LIN {X 0,Y 169.954,Z 453.379,A -85,B 0,C 180,E1 -25767.886,E2 -25767.886} C_VEL
LIN {X 0,Y 165.265,Z 466.004,A -85,B 0,C 180,E1 -25769.338,E2 -25769.338} C_VEL
LIN {X 0,Y 160.143,Z 477.221,A -85,B 0,C 180,E1 -25771.158,E2 -25771.158} C_VEL
LIN {X 0,Y 154.638,Z 487.355,A -85,B 0,C 180,E1 -25773.432,E2 -25773.432} C_VEL
LIN {X 0,Y 148.228,Z 497.15,A -85,B 0,C 180,E1 -25776.293,E2 -25776.293} C_VEL
LIN {X 0,Y 142.57,Z 504.593,A -85,B 0,C 180,E1 -25779.183,E2 -25779.183} C_VEL
LIN {X 0,Y 136.506,Z 511.591,A -85,B 0,C 180,E1 -25782.809,E2 -25782.809} C_VEL
LIN {X 0,Y 129.978,Z 518.044,A -85,B 0,C 180,E1 -25787.48,E2 -25787.48} C_VEL
LIN {X 0,Y 125.036,Z 522.318,A -85,B 0,C 180,E1 -25791.9,E2 -25791.9} C_VEL
LIN {X 0,Y 122.256,Z 524.487,A -85,B 0,C 180,E1 -25794.913,E2 -25794.913} C_VEL
LIN {X 0,Y 119.731,Z 526.212,A -85,B 0,C 180,E1 -25798.113,E2 -25798.113} C_VEL
LIN {X 0,Y 115.834,Z 528.4,A -85,B 0,C 180,E1 -25804.87,E2 -25804.87} C_VEL
LIN {X 0,Y 114.432,Z 528.886,A -85,B 0,C 180,E1 -25808.379,E2 -25808.379} C_VEL
LIN {X 0,Y 113.36,Z 528.935,A -85,B 0,C 180,E1 -25811.944,E2 -25811.944} C_VEL
LIN {X 0,Y 112.313,Z 527.87,A -85,B 0,C 180,E1 -25819.182,E2 -25819.182} C_VEL
LIN {X 0,Y 112.317,Z 526.734,A -85,B 0,C 180,E1 -25822.813,E2 -25822.813} C_VEL
LIN {X 0,Y 112.709,Z 525.151,A -85,B 0,C 180,E1 -25826.427,E2 -25826.427} C_VEL
LIN {X 0,Y 113.499,Z 522.024,A -85,B 0,C 180,E1 -25831.776,E2 -25831.776} C_VEL
LIN {X 0,Y 115.038,Z 517.849,A -85,B 0,C 180,E1 -25837.021,E2 -25837.021} C_VEL
LIN {X 0,Y 117.816,Z 511.498,A -85,B 0,C 180,E1 -25842.928,E2 -25842.928} C_VEL
LIN {X 0,Y 120.909,Z 504.594,A -85,B 0,C 180,E1 -25847.77,E2 -25847.77} C_VEL
LIN {X 0,Y 124.835,Z 495.925,A -85,B 0,C 180,E1 -25852.337,E2 -25852.337} C_VEL
LIN {X 0,Y 128.597,Z 487.054,A -85,B 0,C 180,E1 -25855.928,E2 -25855.928} C_VEL
LIN {X 0,Y 132.376,Z 477.3,A -85,B 0,C 180,E1 -25858.979,E2 -25858.979} C_VEL
LIN {X 0,Y 136.006,Z 466.57,A -85,B 0,C 180,E1 -25861.55,E2 -25861.55} C_VEL
LIN {X 0,Y 139.168,Z 454.593,A -85,B 0,C 180,E1 -25863.747,E2 -25863.747} C_VEL
LIN {X 0,Y 141.844,Z 442.071,A -85,B 0,C 180,E1 -25865.388,E2 -25865.388} C_VEL
LIN {X 0,Y 143.68,Z 429.753,A -85,B 0,C 180,E1 -25866.505,E2 -25866.505} C_VEL
LIN {X 0,Y 144.953,Z 414.737,A -85,B 0,C 180,E1 -25867.3,E2 -25867.3} C_VEL
LIN {X 0,Y 147.183,Z 381.844,A -85,B 0,C 180,E1 -25868.662,E2 -25868.662} C_VEL
LIN {X 0,Y 143.364,Z 373.581,A -85,B 0,C 180,E1 -25870.727,E2 -25870.727} C_VEL
LIN {X 0,Y 138.443,Z 364.416,A -85,B 0,C 180,E1 -25873.568,E2 -25873.568} C_VEL
LIN {X 0,Y 132.527,Z 354.94,A -85,B 0,C 180,E1 -25877.383,E2 -25877.383} C_VEL
LIN {X 0,Y 129.11,Z 350.145,A -85,B 0,C 180,E1 -25879.855,E2 -25879.855} C_VEL
LIN {X 0,Y 126.584,Z 346.535,A -85,B 0,C 180,E1 -25881.884,E2 -25881.884} C_VEL
LIN {X 0,Y 124.126,Z 343.341,A -85,B 0,C 180,E1 -25884.023,E2 -25884.023} C_VEL
LIN {X 0,Y 123.216,Z 342.017,A -85,B 0,C 180,E1 -25884.889,E2 -25884.889} C_VEL
LIN {X 0,Y 120.836,Z 339.591,A -85,B 0,C 180,E1 -25887.204,E2 -25887.204} C_VEL
LIN {X 0,Y 119.433,Z 336.949,A -85,B 0,C 180,E1 -25888.862,E2 -25888.862} C_VEL
LIN {X 0,Y 116.762,Z 335.135,A -85,B 0,C 180,E1 -25891.949,E2 -25891.949} C_VEL
LIN {X 0,Y 115.281,Z 332.838,A -85,B 0,C 180,E1 -25894.132,E2 -25894.132} C_VEL
LIN {X 0,Y 114.896,Z 331.137,A -85,B 0,C 180,E1 -25895.066,E2 -25895.066} C_VEL
LIN {X 0,Y 114.985,Z 331.156,A -85,B 0,C 180,E1 -25898.485,E2 -25898.485} C_VEL
LIN {X 0,Y 115.113,Z 331.108,A -85,B 0,C 180,E1 -25905.864,E2 -25905.864} C_VEL
LIN {X 0,Y 115.315,Z 331.119,A -85,B 0,C 180,E1 -25909.464,E2 -25909.464} C_VEL
LIN {X 0,Y 115.489,Z 331.058,A -85,B 0,C 180,E1 -25916.51,E2 -25916.51} C_VEL
LIN {X 0,Y 115.977,Z 331.035,A -85,B 0,C 180,E1 -25919.999,E2 -25919.999} C_VEL
LIN {X 0,Y 115.35,Z 331.075,A -85,B 0,C 180,E1 -25926.998,E2 -25926.998} C_VEL
LIN {X 0,Y 115.209,Z 331.131,A -85,B 0,C 180,E1 -25932.558,E2 -25932.558} C_VEL
LIN {X 0,Y 115.029,Z 331.167,A -85,B 0,C 180,E1 -25935.617,E2 -25935.617} C_VEL
LIN {X 0,Y 115.766,Z 333.599,A -85,B 0,C 180,E1 -25936.987,E2 -25936.987} C_VEL
LIN {X 0,Y 117.399,Z 335.687,A -85,B 0,C 180,E1 -25939.223,E2 -25939.223} C_VEL
LIN {X 0,Y 119.578,Z 337.12,A -85,B 0,C 180,E1 -25941.67,E2 -25941.67} C_VEL
LIN {X 0,Y 121.212,Z 340.163,A -85,B 0,C 180,E1 -25943.566,E2 -25943.566} C_VEL
LIN {X 0,Y 123.785,Z 342.605,A -85,B 0,C 180,E1 -25945.991,E2 -25945.991} C_VEL
LIN {X 0,Y 126.065,Z 346.012,A -85,B 0,C 180,E1 -25948.058,E2 -25948.058} C_VEL
LIN {X 0,Y 127.461,Z 347.601,A -85,B 0,C 180,E1 -25949.184,E2 -25949.184} C_VEL
LIN {X 0,Y 132.939,Z 355.533,A -85,B 0,C 180,E1 -25953.263,E2 -25953.263} C_VEL
LIN {X 0,Y 135.888,Z 360.462,A -85,B 0,C 180,E1 -25955.238,E2 -25955.238} C_VEL
LIN {X 0,Y 140.904,Z 371.644,A -85,B 0,C 180,E1 -25958.455,E2 -25958.455} C_VEL
LIN {X 0,Y 144.8,Z 382.281,A -85,B 0,C 180,E1 -25960.822,E2 -25960.822} C_VEL
LIN {X 0,Y 145.866,Z 386.133,A -85,B 0,C 180,E1 -25961.495,E2 -25961.495} C_VEL
LIN {X 0,Y 146.293,Z 398.588,A -85,B 0,C 180,E1 -25962.485,E2 -25962.485} C_VEL
LIN {X 0,Y 143.56,Z 436.22,A -85,B 0,C 180,E1 -25964.112,E2 -25964.112} C_VEL
LIN {X 0,Y 141.608,Z 449.705,A -85,B 0,C 180,E1 -25965.163,E2 -25965.163} C_VEL
LIN {X 0,Y 138.867,Z 462.391,A -85,B 0,C 180,E1 -25966.652,E2 -25966.652} C_VEL
LIN {X 0,Y 135.486,Z 474.2,A -85,B 0,C 180,E1 -25968.593,E2 -25968.593} C_VEL
LIN {X 0,Y 131.576,Z 485.585,A -85,B 0,C 180,E1 -25971.123,E2 -25971.123} C_VEL
LIN {X 0,Y 127.594,Z 495.844,A -85,B 0,C 180,E1 -25974.178,E2 -25974.178} C_VEL
LIN {X 0,Y 123.397,Z 505.909,A -85,B 0,C 180,E1 -25978.206,E2 -25978.206} C_VEL
LIN {X 0,Y 120.567,Z 511.911,A -85,B 0,C 180,E1 -25981.194,E2 -25981.194} C_VEL
LIN {X 0,Y 118.406,Z 517.269,A -85,B 0,C 180,E1 -25984.51,E2 -25984.51} C_VEL
LIN {X 0,Y 116.081,Z 522.835,A -85,B 0,C 180,E1 -25988.697,E2 -25988.697} C_VEL
LIN {X 0,Y 113.916,Z 528.259,A -85,B 0,C 180,E1 -25993.879,E2 -25993.879} C_VEL
LIN {X 0,Y 112.782,Z 532.492,A -85,B 0,C 180,E1 -25999.223,E2 -25999.223} C_VEL
LIN {X 0,Y 112.433,Z 534.724,A -85,B 0,C 180,E1 -26002.816,E2 -26002.816} C_VEL
LIN {X 0,Y 112.492,Z 537.26,A -85,B 0,C 180,E1 -26008.387,E2 -26008.387} C_VEL
LIN {X 0,Y 112.47,Z 538.122,A -85,B 0,C 180,E1 -26011.162,E2 -26011.162} C_VEL
LIN {X 0,Y 112.405,Z 539.12,A -85,B 0,C 180,E1 -26017.181,E2 -26017.181} C_VEL
LIN {X 0,Y 113.531,Z 538.827,A -85,B 0,C 180,E1 -26024.334,E2 -26024.334} C_VEL
LIN {X 0,Y 116.284,Z 537.016,A -85,B 0,C 180,E1 -26031.259,E2 -26031.259} C_VEL
LIN {X 0,Y 118.375,Z 535.488,A -85,B 0,C 180,E1 -26034.554,E2 -26034.554} C_VEL
LIN {X 0,Y 122.165,Z 532.423,A -85,B 0,C 180,E1 -26039.272,E2 -26039.272} C_VEL
LIN {X 0,Y 126.661,Z 528.327,A -85,B 0,C 180,E1 -26043.699,E2 -26043.699} C_VEL
LIN {X 0,Y 132.806,Z 522.078,A -85,B 0,C 180,E1 -26048.445,E2 -26048.445} C_VEL
LIN {X 0,Y 138.861,Z 515.309,A -85,B 0,C 180,E1 -26052.111,E2 -26052.111} C_VEL
LIN {X 0,Y 145.542,Z 506.936,A -85,B 0,C 180,E1 -26055.416,E2 -26055.416} C_VEL
LIN {X 0,Y 151.382,Z 498.339,A -85,B 0,C 180,E1 -26057.969,E2 -26057.969} C_VEL
LIN {X 0,Y 153.654,Z 494.853,A -85,B 0,C 180,E1 -26058.768,E2 -26058.768} C_VEL
LIN {X 0,Y 155.897,Z 490.401,A -85,B 0,C 180,E1 -26059.955,E2 -26059.955} C_VEL
LIN {X 0,Y 158.231,Z 482.914,A -85,B 0,C 180,E1 -26062.187,E2 -26062.187} C_VEL
LIN {X 0,Y 160.346,Z 474.972,A -85,B 0,C 180,E1 -26064.172,E2 -26064.172} C_VEL
LIN {X 0,Y 162.147,Z 469.815,A -85,B 0,C 180,E1 -26064.959,E2 -26064.959} C_VEL
LIN {X 0,Y 166.612,Z 457.272,A -85,B 0,C 180,E1 -26066.142,E2 -26066.142} C_VEL
LIN {X 0,Y 169.968,Z 444.445,A -85,B 0,C 180,E1 -26066.992,E2 -26066.992} C_VEL
LIN {X 0,Y 172.089,Z 431.144,A -85,B 0,C 180,E1 -26067.598,E2 -26067.598} C_VEL
LIN {X 0,Y 173.3,Z 418.29,A -85,B 0,C 180,E1 -26068.013,E2 -26068.013} C_VEL
LIN {X 0,Y 170.042,Z 408.838,A -85,B 0,C 180,E1 -26071.06,E2 -26071.06} C_VEL
LIN {X 0,Y 166.847,Z 400.851,A -85,B 0,C 180,E1 -26074.424,E2 -26074.424} C_VEL
LIN {X 0,Y 164.442,Z 395.255,A -85,B 0,C 180,E1 -26077.379,E2 -26077.379} C_VEL
LIN {X 0,Y 161.996,Z 390.005,A -85,B 0,C 180,E1 -26081.012,E2 -26081.012} C_VEL
LIN {X 0,Y 159.926,Z 386.674,A -85,B 0,C 180,E1 -26084.859,E2 -26084.859} C_VEL
LIN {X 0,Y 159.509,Z 385.905,A -85,B 0,C 180,E1 -26085.846,E2 -26085.846} C_VEL
LIN {X 0,Y 157.79,Z 383.124,A -85,B 0,C 180,E1 -26091.856,E2 -26091.856} C_VEL
LIN {X 0,Y 157.642,Z 381.317,A -85,B 0,C 180,E1 -26094.885,E2 -26094.885} C_VEL
LIN {X 0,Y 157.697,Z 381.298,A -85,B 0,C 180,E1 -26097.59,E2 -26097.59} C_VEL
LIN {X 0,Y 158.291,Z 384.205,A -85,B 0,C 180,E1 -26102.307,E2 -26102.307} C_VEL
LIN {X 0,Y 159.882,Z 386.192,A -85,B 0,C 180,E1 -26106.627,E2 -26106.627} C_VEL
LIN {X 0,Y 161.996,Z 389.909,A -85,B 0,C 180,E1 -26110.649,E2 -26110.649} C_VEL
LIN {X 0,Y 165.028,Z 395.159,A -85,B 0,C 180,E1 -26114.884,E2 -26114.884} C_VEL
LIN {X 0,Y 168.167,Z 400.686,A -85,B 0,C 180,E1 -26118.346,E2 -26118.346} C_VEL
LIN {X 0,Y 172.368,Z 408.93,A -85,B 0,C 180,E1 -26122.237,E2 -26122.237} C_VEL
LIN {X 0,Y 173.842,Z 412.055,A -85,B 0,C 180,E1 -26123.463,E2 -26123.463} C_VEL
LIN {X 0,Y 171.856,Z 429.918,A -85,B 0,C 180,E1 -26124.078,E2 -26124.078} C_VEL
LIN {X 0,Y 169.4,Z 442.515,A -85,B 0,C 180,E1 -26124.856,E2 -26124.856} C_VEL
LIN {X 0,Y 165.916,Z 454.623,A -85,B 0,C 180,E1 -26125.912,E2 -26125.912} C_VEL
LIN {X 0,Y 161.171,Z 466.872,A -85,B 0,C 180,E1 -26127.322,E2 -26127.322} C_VEL
LIN {X 0,Y 155.877,Z 477.959,A -85,B 0,C 180,E1 -26129.129,E2 -26129.129} C_VEL
LIN {X 0,Y 150.482,Z 487.489,A -85,B 0,C 180,E1 -26131.254,E2 -26131.254} C_VEL
LIN {X 0,Y 144.072,Z 496.935,A -85,B 0,C 180,E1 -26133.979,E2 -26133.979} C_VEL
LIN {X 0,Y 138.219,Z 504.334,A -85,B 0,C 180,E1 -26136.793,E2 -26136.793} C_VEL
LIN {X 0,Y 132.466,Z 510.715,A -85,B 0,C 180,E1 -26139.988,E2 -26139.988} C_VEL
LIN {X 0,Y 126.633,Z 516.425,A -85,B 0,C 180,E1 -26143.826,E2 -26143.826} C_VEL
LIN {X 0,Y 121.169,Z 521.105,A -85,B 0,C 180,E1 -26148.165,E2 -26148.165} C_VEL
LIN {X 0,Y 116.381,Z 524.643,A -85,B 0,C 180,E1 -26152.855,E2 -26152.855} C_VEL
LIN {X 0,Y 113.63,Z 526.425,A -85,B 0,C 180,E1 -26156.178,E2 -26156.178} C_VEL
LIN {X 0,Y 109.315,Z 528.668,A -85,B 0,C 180,E1 -26163.256,E2 -26163.256} C_VEL
LIN {X 0,Y 107.754,Z 529.194,A -85,B 0,C 180,E1 -26166.965,E2 -26166.965} C_VEL
LIN {X 0,Y 106.525,Z 529.284,A -85,B 0,C 180,E1 -26170.741,E2 -26170.741} C_VEL
LIN {X 0,Y 105.254,Z 528.274,A -85,B 0,C 180,E1 -26178.447,E2 -26178.447} C_VEL
LIN {X 0,Y 105.214,Z 527.182,A -85,B 0,C 180,E1 -26182.325,E2 -26182.325} C_VEL
LIN {X 0,Y 105.622,Z 525.499,A -85,B 0,C 180,E1 -26186.473,E2 -26186.473} C_VEL
LIN {X 0,Y 106.413,Z 522.565,A -85,B 0,C 180,E1 -26191.895,E2 -26191.895} C_VEL
LIN {X 0,Y 107.983,Z 518.455,A -85,B 0,C 180,E1 -26197.482,E2 -26197.482} C_VEL
LIN {X 0,Y 110.91,Z 512.171,A -85,B 0,C 180,E1 -26203.749,E2 -26203.749} C_VEL
LIN {X 0,Y 114.193,Z 505.347,A -85,B 0,C 180,E1 -26208.853,E2 -26208.853} C_VEL
LIN {X 0,Y 118.337,Z 496.805,A -85,B 0,C 180,E1 -26213.636,E2 -26213.636} C_VEL
LIN {X 0,Y 122.271,Z 488.046,A -85,B 0,C 180,E1 -26217.379,E2 -26217.379} C_VEL
LIN {X 0,Y 126.71,Z 477.255,A -85,B 0,C 180,E1 -26220.87,E2 -26220.87} C_VEL
LIN {X 0,Y 130.528,Z 466.399,A -85,B 0,C 180,E1 -26223.499,E2 -26223.499} C_VEL
LIN {X 0,Y 133.872,Z 454.288,A -85,B 0,C 180,E1 -26225.737,E2 -26225.737} C_VEL
LIN {X 0,Y 136.679,Z 441.562,A -85,B 0,C 180,E1 -26227.404,E2 -26227.404} C_VEL
LIN {X 0,Y 138.605,Z 428.722,A -85,B 0,C 180,E1 -26228.527,E2 -26228.527} C_VEL
LIN {X 0,Y 140.024,Z 411.792,A -85,B 0,C 180,E1 -26229.383,E2 -26229.383} C_VEL
LIN {X 0,Y 141.986,Z 384.117,A -85,B 0,C 180,E1 -26230.548,E2 -26230.548} C_VEL
LIN {X 0,Y 136.478,Z 372.568,A -85,B 0,C 180,E1 -26233.867,E2 -26233.867} C_VEL
LIN {X 0,Y 131.079,Z 363.313,A -85,B 0,C 180,E1 -26237.464,E2 -26237.464} C_VEL
LIN {X 0,Y 126.527,Z 356.335,A -85,B 0,C 180,E1 -26240.933,E2 -26240.933} C_VEL
LIN {X 0,Y 123.686,Z 352.328,A -85,B 0,C 180,E1 -26243.37,E2 -26243.37} C_VEL
LIN {X 0,Y 120.776,Z 348.238,A -85,B 0,C 180,E1 -26246.188,E2 -26246.188} C_VEL
LIN {X 0,Y 118.216,Z 345.2,A -85,B 0,C 180,E1 -26248.944,E2 -26248.944} C_VEL
LIN {X 0,Y 117.162,Z 343.409,A -85,B 0,C 180,E1 -26250.275,E2 -26250.275} C_VEL
LIN {X 0,Y 114.737,Z 341.346,A -85,B 0,C 180,E1 -26253.389,E2 -26253.389} C_VEL
LIN {X 0,Y 113.179,Z 338.5,A -85,B 0,C 180,E1 -26256.004,E2 -26256.004} C_VEL
LIN {X 0,Y 112.812,Z 337.909,A -85,B 0,C 180,E1 -26256.666,E2 -26256.666} C_VEL
LIN {X 0,Y 109.796,Z 335.963,A -85,B 0,C 180,E1 -26262.779,E2 -26262.779} C_VEL
LIN {X 0,Y 108.452,Z 333.244,A -85,B 0,C 180,E1 -26267.91,E2 -26267.91} C_VEL
LIN {X 0,Y 108.274,Z 331.996,A -85,B 0,C 180,E1 -26269.716,E2 -26269.716} C_VEL
LIN {X 0,Y 108.902,Z 331.915,A -85,B 0,C 180,E1 -26279.999,E2 -26279.999} C_VEL
LIN {X 0,Y 108.583,Z 332.143,A -85,B 0,C 180,E1 -26282.433,E2 -26282.433} C_VEL
LIN {X 0,Y 108.955,Z 334.021,A -85,B 0,C 180,E1 -26284.624,E2 -26284.624} C_VEL
LIN {X 0,Y 111.057,Z 336.803,A -85,B 0,C 180,E1 -26290.482,E2 -26290.482} C_VEL
LIN {X 0,Y 113.226,Z 338.186,A -85,B 0,C 180,E1 -26294.375,E2 -26294.375} C_VEL
LIN {X 0,Y 114.698,Z 341.256,A -85,B 0,C 180,E1 -26296.92,E2 -26296.92} C_VEL
LIN {X 0,Y 117.543,Z 343.903,A -85,B 0,C 180,E1 -26300.564,E2 -26300.564} C_VEL
LIN {X 0,Y 119.702,Z 347.229,A -85,B 0,C 180,E1 -26303.098,E2 -26303.098} C_VEL
LIN {X 0,Y 121.442,Z 349.031,A -85,B 0,C 180,E1 -26304.835,E2 -26304.835} C_VEL
LIN {X 0,Y 124.045,Z 352.644,A -85,B 0,C 180,E1 -26307.294,E2 -26307.294} C_VEL
LIN {X 0,Y 128.199,Z 358.783,A -85,B 0,C 180,E1 -26310.755,E2 -26310.755} C_VEL
LIN {X 0,Y 131.886,Z 364.746,A -85,B 0,C 180,E1 -26313.477,E2 -26313.477} C_VEL
LIN {X 0,Y 136.397,Z 375.036,A -85,B 0,C 180,E1 -26316.653,E2 -26316.653} C_VEL
LIN {X 0,Y 140.213,Z 385.883,A -85,B 0,C 180,E1 -26319.199,E2 -26319.199} C_VEL
LIN {X 0,Y 140.883,Z 388.479,A -85,B 0,C 180,E1 -26319.67,E2 -26319.67} C_VEL
LIN {X 0,Y 141.103,Z 399.609,A -85,B 0,C 180,E1 -26320.555,E2 -26320.555} C_VEL
LIN {X 0,Y 138.379,Z 435.693,A -85,B 0,C 180,E1 -26322.145,E2 -26322.145} C_VEL
LIN {X 0,Y 136.308,Z 449.382,A -85,B 0,C 180,E1 -26323.218,E2 -26323.218} C_VEL
LIN {X 0,Y 133.493,Z 461.901,A -85,B 0,C 180,E1 -26324.703,E2 -26324.703} C_VEL
LIN {X 0,Y 130.223,Z 472.946,A -85,B 0,C 180,E1 -26326.517,E2 -26326.517} C_VEL
LIN {X 0,Y 126.133,Z 484.507,A -85,B 0,C 180,E1 -26329.101,E2 -26329.101} C_VEL
LIN {X 0,Y 121.913,Z 494.927,A -85,B 0,C 180,E1 -26332.227,E2 -26332.227} C_VEL
LIN {X 0,Y 118.145,Z 503.441,A -85,B 0,C 180,E1 -26335.587,E2 -26335.587} C_VEL
LIN {X 0,Y 113.695,Z 512.647,A -85,B 0,C 180,E1 -26340.36,E2 -26340.36} C_VEL
LIN {X 0,Y 111.401,Z 517.812,A -85,B 0,C 180,E1 -26343.791,E2 -26343.791} C_VEL
LIN {X 0,Y 108.521,Z 524.19,A -85,B 0,C 180,E1 -26349.131,E2 -26349.131} C_VEL
LIN {X 0,Y 106.527,Z 529.254,A -85,B 0,C 180,E1 -26354.696,E2 -26354.696} C_VEL
LIN {X 0,Y 105.532,Z 533.167,A -85,B 0,C 180,E1 -26360.414,E2 -26360.414} C_VEL
LIN {X 0,Y 105.32,Z 536.026,A -85,B 0,C 180,E1 -26366.171,E2 -26366.171} C_VEL
LIN {X 0,Y 105.431,Z 537.605,A -85,B 0,C 180,E1 -26370.856,E2 -26370.856} C_VEL
LIN {X 0,Y 105.334,Z 538.761,A -85,B 0,C 180,E1 -26377.666,E2 -26377.666} C_VEL
LIN {X 0,Y 105.769,Z 538.844,A -85,B 0,C 180,E1 -26381.496,E2 -26381.496} C_VEL
LIN {X 0,Y 107.904,Z 537.837,A -85,B 0,C 180,E1 -26389.003,E2 -26389.003} C_VEL
LIN {X 0,Y 109.684,Z 536.767,A -85,B 0,C 180,E1 -26392.607,E2 -26392.607} C_VEL
LIN {X 0,Y 111.941,Z 535.286,A -85,B 0,C 180,E1 -26396.068,E2 -26396.068} C_VEL
LIN {X 0,Y 116.011,Z 532.268,A -85,B 0,C 180,E1 -26400.99,E2 -26400.99} C_VEL
LIN {X 0,Y 120.794,Z 528.222,A -85,B 0,C 180,E1 -26405.576,E2 -26405.576} C_VEL
LIN {X 0,Y 127.306,Z 522.046,A -85,B 0,C 180,E1 -26410.439,E2 -26410.439} C_VEL
LIN {X 0,Y 133.678,Z 515.346,A -85,B 0,C 180,E1 -26414.153,E2 -26414.153} C_VEL
LIN {X 0,Y 140.657,Z 507.06,A -85,B 0,C 180,E1 -26417.473,E2 -26417.473} C_VEL
LIN {X 0,Y 146.735,Z 498.585,A -85,B 0,C 180,E1 -26420.023,E2 -26420.023} C_VEL
LIN {X 0,Y 153.27,Z 488.129,A -85,B 0,C 180,E1 -26422.274,E2 -26422.274} C_VEL
LIN {X 0,Y 159.292,Z 476.387,A -85,B 0,C 180,E1 -26424.162,E2 -26424.162} C_VEL
LIN {X 0,Y 162.147,Z 469.815,A -85,B 0,C 180,E1 -26424.959,E2 -26424.959} C_VEL
LIN {X 0,Y 163.869,Z 464.575,A -85,B 0,C 180,E1 -26425.674,E2 -26425.674} C_VEL
LIN {X 0,Y 165.34,Z 455.878,A -85,B 0,C 180,E1 -26427.273,E2 -26427.273} C_VEL
LIN {X 0,Y 166.335,Z 446.985,A -85,B 0,C 180,E1 -26428.752,E2 -26428.752} C_VEL
LIN {X 0,Y 167.207,Z 441.344,A -85,B 0,C 180,E1 -26429.277,E2 -26429.277} C_VEL
LIN {X 0,Y 169.186,Z 428.054,A -85,B 0,C 180,E1 -26429.805,E2 -26429.805} C_VEL
LIN {X 0,Y 169.798,Z 421.095,A -85,B 0,C 180,E1 -26430.049,E2 -26430.049} C_VEL
LIN {X 0,Y 167.122,Z 413.122,A -85,B 0,C 180,E1 -26432.835,E2 -26432.835} C_VEL
LIN {X 0,Y 164.516,Z 406.154,A -85,B 0,C 180,E1 -26435.899,E2 -26435.899} C_VEL
LIN {X 0,Y 162.539,Z 401.124,A -85,B 0,C 180,E1 -26438.604,E2 -26438.604} C_VEL
LIN {X 0,Y 160.748,Z 396.858,A -85,B 0,C 180,E1 -26441.521,E2 -26441.521} C_VEL
LIN {X 0,Y 158.687,Z 393.329,A -85,B 0,C 180,E1 -26445.628,E2 -26445.628} C_VEL
LIN {X 0,Y 156.786,Z 389.519,A -85,B 0,C 180,E1 -26453.162,E2 -26453.162} C_VEL
LIN {X 0,Y 156.768,Z 388.418,A -85,B 0,C 180,E1 -26454.857,E2 -26454.857} C_VEL
LIN {X 0,Y 156.798,Z 388.676,A -85,B 0,C 180,E1 -26457.721,E2 -26457.721} C_VEL
LIN {X 0,Y 157.349,Z 391.227,A -85,B 0,C 180,E1 -26462.08,E2 -26462.08} C_VEL
LIN {X 0,Y 158.686,Z 392.968,A -85,B 0,C 180,E1 -26465.959,E2 -26465.959} C_VEL
LIN {X 0,Y 160.613,Z 396.596,A -85,B 0,C 180,E1 -26469.922,E2 -26469.922} C_VEL
LIN {X 0,Y 163.22,Z 401.372,A -85,B 0,C 180,E1 -26473.859,E2 -26473.859} C_VEL
LIN {X 0,Y 166.248,Z 407.044,A -85,B 0,C 180,E1 -26477.451,E2 -26477.451} C_VEL
LIN {X 0,Y 169.878,Z 414.594,A -85,B 0,C 180,E1 -26481.065,E2 -26481.065} C_VEL
LIN {X 0,Y 170.319,Z 415.597,A -85,B 0,C 180,E1 -26481.47,E2 -26481.47} C_VEL
LIN {X 0,Y 168.485,Z 430.752,A -85,B 0,C 180,E1 -26481.993,E2 -26481.993} C_VEL
LIN {X 0,Y 166.155,Z 442.266,A -85,B 0,C 180,E1 -26482.683,E2 -26482.683} C_VEL
LIN {X 0,Y 162.705,Z 454.172,A -85,B 0,C 180,E1 -26483.691,E2 -26483.691} C_VEL
LIN {X 0,Y 157.991,Z 466.137,A -85,B 0,C 180,E1 -26484.998,E2 -26484.998} C_VEL
LIN {X 0,Y 152.463,Z 477.464,A -85,B 0,C 180,E1 -26486.736,E2 -26486.736} C_VEL
LIN {X 0,Y 147.179,Z 486.632,A -85,B 0,C 180,E1 -26488.694,E2 -26488.694} C_VEL
LIN {X 0,Y 141.422,Z 495.073,A -85,B 0,C 180,E1 -26490.995,E2 -26490.995} C_VEL
LIN {X 0,Y 133.998,Z 504.211,A -85,B 0,C 180,E1 -26494.307,E2 -26494.307} C_VEL
LIN {X 0,Y 127.662,Z 510.948,A -85,B 0,C 180,E1 -26497.66,E2 -26497.66} C_VEL
LIN {X 0,Y 121.717,Z 516.455,A -85,B 0,C 180,E1 -26501.359,E2 -26501.359} C_VEL
LIN {X 0,Y 115.868,Z 521.2,A -85,B 0,C 180,E1 -26505.773,E2 -26505.773} C_VEL
LIN {X 0,Y 110.675,Z 524.8,A -85,B 0,C 180,E1 -26510.582,E2 -26510.582} C_VEL
LIN {X 0,Y 107.673,Z 526.635,A -85,B 0,C 180,E1 -26514.027,E2 -26514.027} C_VEL
LIN {X 0,Y 105.09,Z 527.989,A -85,B 0,C 180,E1 -26517.659,E2 -26517.659} C_VEL
LIN {X 0,Y 101.126,Z 529.491,A -85,B 0,C 180,E1 -26525.359,E2 -26525.359} C_VEL
LIN {X 0,Y 99.751,Z 529.633,A -85,B 0,C 180,E1 -26529.376,E2 -26529.376} C_VEL
LIN {X 0,Y 98.228,Z 528.675,A -85,B 0,C 180,E1 -26537.608,E2 -26537.608} C_VEL
LIN {X 0,Y 98.097,Z 527.616,A -85,B 0,C 180,E1 -26541.765,E2 -26541.765} C_VEL
LIN {X 0,Y 98.557,Z 525.764,A -85,B 0,C 180,E1 -26546.712,E2 -26546.712} C_VEL
LIN {X 0,Y 99.731,Z 521.863,A -85,B 0,C 180,E1 -26554.044,E2 -26554.044} C_VEL
LIN {X 0,Y 101.753,Z 517.439,A -85,B 0,C 180,E1 -26559.946,E2 -26559.946} C_VEL
LIN {X 0,Y 105.149,Z 510.753,A -85,B 0,C 180,E1 -26566.505,E2 -26566.505} C_VEL
LIN {X 0,Y 108.885,Z 503.473,A -85,B 0,C 180,E1 -26571.788,E2 -26571.788} C_VEL
LIN {X 0,Y 113.48,Z 494.433,A -85,B 0,C 180,E1 -26576.682,E2 -26576.682} C_VEL
LIN {X 0,Y 117.886,Z 485.043,A -85,B 0,C 180,E1 -26580.45,E2 -26580.45} C_VEL
LIN {X 0,Y 122.224,Z 474.617,A -85,B 0,C 180,E1 -26583.606,E2 -26583.606} C_VEL
LIN {X 0,Y 126.236,Z 463.054,A -85,B 0,C 180,E1 -26586.268,E2 -26586.268} C_VEL
LIN {X 0,Y 129.511,Z 450.815,A -85,B 0,C 180,E1 -26588.367,E2 -26588.367} C_VEL
LIN {X 0,Y 132.217,Z 437.848,A -85,B 0,C 180,E1 -26589.892,E2 -26589.892} C_VEL
LIN {X 0,Y 133.947,Z 425.431,A -85,B 0,C 180,E1 -26590.857,E2 -26590.857} C_VEL
LIN {X 0,Y 136.935,Z 386.564,A -85,B 0,C 180,E1 -26592.563,E2 -26592.563} C_VEL
LIN {X 0,Y 131.771,Z 375.641,A -85,B 0,C 180,E1 -26596.008,E2 -26596.008} C_VEL
LIN {X 0,Y 126.211,Z 366.056,A -85,B 0,C 180,E1 -26600.179,E2 -26600.179} C_VEL
LIN {X 0,Y 122.912,Z 361,A -85,B 0,C 180,E1 -26603.007,E2 -26603.007} C_VEL
LIN {X 0,Y 120.861,Z 357.996,A -85,B 0,C 180,E1 -26604.953,E2 -26604.953} C_VEL
LIN {X 0,Y 118.401,Z 354.377,A -85,B 0,C 180,E1 -26607.551,E2 -26607.551} C_VEL
LIN {X 0,Y 115.938,Z 351.149,A -85,B 0,C 180,E1 -26610.461,E2 -26610.461} C_VEL
LIN {X 0,Y 115.149,Z 349.933,A -85,B 0,C 180,E1 -26611.52,E2 -26611.52} C_VEL
LIN {X 0,Y 112.655,Z 347.357,A -85,B 0,C 180,E1 -26615.095,E2 -26615.095} C_VEL
LIN {X 0,Y 111.258,Z 344.739,A -85,B 0,C 180,E1 -26617.726,E2 -26617.726} C_VEL
LIN {X 0,Y 108.256,Z 342.333,A -85,B 0,C 180,E1 -26624.707,E2 -26624.707} C_VEL
LIN {X 0,Y 107.247,Z 339.027,A -85,B 0,C 180,E1 -26630.38,E2 -26630.38} C_VEL
LIN {X 0,Y 107.423,Z 338.911,A -85,B 0,C 180,E1 -26640.936,E2 -26640.936} C_VEL
LIN {X 0,Y 108.358,Z 341.954,A -85,B 0,C 180,E1 -26645.816,E2 -26645.816} C_VEL
LIN {X 0,Y 111.096,Z 344.552,A -85,B 0,C 180,E1 -26652.327,E2 -26652.327} C_VEL
LIN {X 0,Y 111.666,Z 345.136,A -85,B 0,C 180,E1 -26653.378,E2 -26653.378} C_VEL
LIN {X 0,Y 113.332,Z 348.228,A -85,B 0,C 180,E1 -26656.348,E2 -26656.348} C_VEL
LIN {X 0,Y 115.528,Z 350.378,A -85,B 0,C 180,E1 -26659.344,E2 -26659.344} C_VEL
LIN {X 0,Y 117.939,Z 353.957,A -85,B 0,C 180,E1 -26662.326,E2 -26662.326} C_VEL
LIN {X 0,Y 119.239,Z 355.523,A -85,B 0,C 180,E1 -26663.723,E2 -26663.723} C_VEL
LIN {X 0,Y 122.511,Z 360.254,A -85,B 0,C 180,E1 -26666.971,E2 -26666.971} C_VEL
LIN {X 0,Y 126.762,Z 366.905,A -85,B 0,C 180,E1 -26670.622,E2 -26670.622} C_VEL
LIN {X 0,Y 128.928,Z 370.958,A -85,B 0,C 180,E1 -26672.336,E2 -26672.336} C_VEL
LIN {X 0,Y 133.239,Z 381.831,A -85,B 0,C 180,E1 -26675.64,E2 -26675.64} C_VEL
LIN {X 0,Y 135.961,Z 390.234,A -85,B 0,C 180,E1 -26677.633,E2 -26677.633} C_VEL
LIN {X 0,Y 136.145,Z 399.898,A -85,B 0,C 180,E1 -26678.458,E2 -26678.458} C_VEL
LIN {X 0,Y 133.375,Z 434.735,A -85,B 0,C 180,E1 -26679.985,E2 -26679.985} C_VEL
LIN {X 0,Y 131.434,Z 447.76,A -85,B 0,C 180,E1 -26681.007,E2 -26681.007} C_VEL
LIN {X 0,Y 128.572,Z 460.292,A -85,B 0,C 180,E1 -26682.441,E2 -26682.441} C_VEL
LIN {X 0,Y 125.094,Z 471.659,A -85,B 0,C 180,E1 -26684.246,E2 -26684.246} C_VEL
LIN {X 0,Y 120.848,Z 483.413,A -85,B 0,C 180,E1 -26686.893,E2 -26686.893} C_VEL
LIN {X 0,Y 116.834,Z 492.884,A -85,B 0,C 180,E1 -26689.708,E2 -26689.708} C_VEL
LIN {X 0,Y 112.294,Z 502.587,A -85,B 0,C 180,E1 -26693.516,E2 -26693.516} C_VEL
LIN {X 0,Y 108.499,Z 510.072,A -85,B 0,C 180,E1 -26697.359,E2 -26697.359} C_VEL
LIN {X 0,Y 105.047,Z 517.13,A -85,B 0,C 180,E1 -26702.072,E2 -26702.072} C_VEL
LIN {X 0,Y 101.881,Z 523.593,A -85,B 0,C 180,E1 -26707.701,E2 -26707.701} C_VEL
LIN {X 0,Y 99.653,Z 528.713,A -85,B 0,C 180,E1 -26713.612,E2 -26713.612} C_VEL
LIN {X 0,Y 98.505,Z 532.68,A -85,B 0,C 180,E1 -26719.723,E2 -26719.723} C_VEL
LIN {X 0,Y 98.227,Z 535.589,A -85,B 0,C 180,E1 -26725.894,E2 -26725.894} C_VEL
LIN {X 0,Y 98.394,Z 537.073,A -85,B 0,C 180,E1 -26730.457,E2 -26730.457} C_VEL
LIN {X 0,Y 98.283,Z 538.395,A -85,B 0,C 180,E1 -26738.22,E2 -26738.22} C_VEL
LIN {X 0,Y 98.784,Z 538.522,A -85,B 0,C 180,E1 -26742.321,E2 -26742.321} C_VEL
LIN {X 0,Y 101.18,Z 537.564,A -85,B 0,C 180,E1 -26750.32,E2 -26750.32} C_VEL
LIN {X 0,Y 105.583,Z 535.082,A -85,B 0,C 180,E1 -26757.769,E2 -26757.769} C_VEL
LIN {X 0,Y 109.973,Z 532.104,A -85,B 0,C 180,E1 -26762.899,E2 -26762.899} C_VEL
LIN {X 0,Y 115.072,Z 528.107,A -85,B 0,C 180,E1 -26767.641,E2 -26767.641} C_VEL
LIN {X 0,Y 121.983,Z 522.015,A -85,B 0,C 180,E1 -26772.605,E2 -26772.605} C_VEL
LIN {X 0,Y 128.686,Z 515.382,A -85,B 0,C 180,E1 -26776.352,E2 -26776.352} C_VEL
LIN {X 0,Y 135.966,Z 507.173,A -85,B 0,C 180,E1 -26779.675,E2 -26779.675} C_VEL
LIN {X 0,Y 142.291,Z 498.801,A -85,B 0,C 180,E1 -26782.207,E2 -26782.207} C_VEL
LIN {X 0,Y 149.052,Z 488.498,A -85,B 0,C 180,E1 -26784.422,E2 -26784.422} C_VEL
LIN {X 0,Y 155.262,Z 476.905,A -85,B 0,C 180,E1 -26786.276,E2 -26786.276} C_VEL
LIN {X 0,Y 160.264,Z 465.448,A -85,B 0,C 180,E1 -26787.579,E2 -26787.579} C_VEL
LIN {X 0,Y 164.588,Z 452.314,A -85,B 0,C 180,E1 -26788.648,E2 -26788.648} C_VEL
LIN {X 0,Y 167.207,Z 441.344,A -85,B 0,C 180,E1 -26789.277,E2 -26789.277} C_VEL
LIN {X 0,Y 167.707,Z 437.557,A -85,B 0,C 180,E1 -26789.591,E2 -26789.591} C_VEL
LIN {X 0,Y 167.666,Z 432.139,A -85,B 0,C 180,E1 -26790.401,E2 -26790.401} C_VEL
LIN {X 0,Y 166.648,Z 425.58,A -85,B 0,C 180,E1 -26791.931,E2 -26791.931} C_VEL
LIN {X 0,Y 165.486,Z 421.091,A -85,B 0,C 180,E1 -26793.329,E2 -26793.329} C_VEL
LIN {X 0,Y 163.809,Z 415.641,A -85,B 0,C 180,E1 -26795.392,E2 -26795.392} C_VEL
LIN {X 0,Y 161.193,Z 408.31,A -85,B 0,C 180,E1 -26799.086,E2 -26799.086} C_VEL
LIN {X 0,Y 159.363,Z 403.562,A -85,B 0,C 180,E1 -26802.284,E2 -26802.284} C_VEL
LIN {X 0,Y 157.346,Z 399.749,A -85,B 0,C 180,E1 -26806.767,E2 -26806.767} C_VEL
LIN {X 0,Y 155.9,Z 396.76,A -85,B 0,C 180,E1 -26813.107,E2 -26813.107} C_VEL
LIN {X 0,Y 155.876,Z 395.665,A -85,B 0,C 180,E1 -26814.827,E2 -26814.827} C_VEL
LIN {X 0,Y 155.901,Z 395.935,A -85,B 0,C 180,E1 -26817.708,E2 -26817.708} C_VEL
LIN {X 0,Y 156.597,Z 398.54,A -85,B 0,C 180,E1 -26822.573,E2 -26822.573} C_VEL
LIN {X 0,Y 157.566,Z 399.911,A -85,B 0,C 180,E1 -26825.44,E2 -26825.44} C_VEL
LIN {X 0,Y 159.778,Z 404.344,A -85,B 0,C 180,E1 -26830.134,E2 -26830.134} C_VEL
LIN {X 0,Y 162.003,Z 408.674,A -85,B 0,C 180,E1 -26833.565,E2 -26833.565} C_VEL
LIN {X 0,Y 164.687,Z 414.087,A -85,B 0,C 180,E1 -26836.902,E2 -26836.902} C_VEL
LIN {X 0,Y 166.97,Z 419.091,A -85,B 0,C 180,E1 -26839.359,E2 -26839.359} C_VEL
LIN {X 0,Y 165.171,Z 432.681,A -85,B 0,C 180,E1 -26839.902,E2 -26839.902} C_VEL
LIN {X 0,Y 162.154,Z 445.813,A -85,B 0,C 180,E1 -26840.719,E2 -26840.719} C_VEL
LIN {X 0,Y 158.019,Z 458.409,A -85,B 0,C 180,E1 -26841.814,E2 -26841.814} C_VEL
LIN {X 0,Y 152.9,Z 470.057,A -85,B 0,C 180,E1 -26843.182,E2 -26843.182} C_VEL
LIN {X 0,Y 147.252,Z 480.606,A -85,B 0,C 180,E1 -26844.933,E2 -26844.933} C_VEL
LIN {X 0,Y 140.502,Z 491.214,A -85,B 0,C 180,E1 -26847.397,E2 -26847.397} C_VEL
LIN {X 0,Y 133.897,Z 499.727,A -85,B 0,C 180,E1 -26850,E2 -26850} C_VEL
LIN {X 0,Y 126.321,Z 507.996,A -85,B 0,C 180,E1 -26853.436,E2 -26853.436} C_VEL
LIN {X 0,Y 119.301,Z 514.616,A -85,B 0,C 180,E1 -26857.322,E2 -26857.322} C_VEL
LIN {X 0,Y 112.794,Z 519.85,A -85,B 0,C 180,E1 -26861.612,E2 -26861.612} C_VEL
LIN {X 0,Y 107.178,Z 523.727,A -85,B 0,C 180,E1 -26866.164,E2 -26866.164} C_VEL
LIN {X 0,Y 101.889,Z 526.83,A -85,B 0,C 180,E1 -26871.629,E2 -26871.629} C_VEL
LIN {X 0,Y 99.024,Z 528.231,A -85,B 0,C 180,E1 -26875.408,E2 -26875.408} C_VEL
LIN {X 0,Y 94.592,Z 529.787,A -85,B 0,C 180,E1 -26883.529,E2 -26883.529} C_VEL
LIN {X 0,Y 93.025,Z 529.974,A -85,B 0,C 180,E1 -26887.809,E2 -26887.809} C_VEL
LIN {X 0,Y 91.195,Z 529.079,A -85,B 0,C 180,E1 -26896.635,E2 -26896.635} C_VEL
LIN {X 0,Y 91.015,Z 528.043,A -85,B 0,C 180,E1 -26901.119,E2 -26901.119} C_VEL
LIN {X 0,Y 91.484,Z 525.986,A -85,B 0,C 180,E1 -26907.091,E2 -26907.091} C_VEL
LIN {X 0,Y 92.665,Z 522.398,A -85,B 0,C 180,E1 -26914.352,E2 -26914.352} C_VEL
LIN {X 0,Y 94.77,Z 518.037,A -85,B 0,C 180,E1 -26920.687,E2 -26920.687} C_VEL
LIN {X 0,Y 97.769,Z 512.495,A -85,B 0,C 180,E1 -26926.713,E2 -26926.713} C_VEL
LIN {X 0,Y 101.611,Z 505.59,A -85,B 0,C 180,E1 -26932.362,E2 -26932.362} C_VEL
LIN {X 0,Y 106.324,Z 496.928,A -85,B 0,C 180,E1 -26937.564,E2 -26937.564} C_VEL
LIN {X 0,Y 110.866,Z 488.05,A -85,B 0,C 180,E1 -26941.535,E2 -26941.535} C_VEL
LIN {X 0,Y 115.322,Z 478.297,A -85,B 0,C 180,E1 -26944.846,E2 -26944.846} C_VEL
LIN {X 0,Y 119.574,Z 467.566,A -85,B 0,C 180,E1 -26947.577,E2 -26947.577} C_VEL
LIN {X 0,Y 123.27,Z 455.592,A -85,B 0,C 180,E1 -26949.899,E2 -26949.899} C_VEL
LIN {X 0,Y 126.351,Z 443.078,A -85,B 0,C 180,E1 -26951.608,E2 -26951.608} C_VEL
LIN {X 0,Y 128.488,Z 430.692,A -85,B 0,C 180,E1 -26952.769,E2 -26952.769} C_VEL
LIN {X 0,Y 130.068,Z 414.573,A -85,B 0,C 180,E1 -26953.631,E2 -26953.631} C_VEL
LIN {X 0,Y 132.061,Z 389.145,A -85,B 0,C 180,E1 -26954.72,E2 -26954.72} C_VEL
LIN {X 0,Y 127.805,Z 379.943,A -85,B 0,C 180,E1 -26957.868,E2 -26957.868} C_VEL
LIN {X 0,Y 123.21,Z 371.639,A -85,B 0,C 180,E1 -26961.656,E2 -26961.656} C_VEL
LIN {X 0,Y 118.947,Z 364.706,A -85,B 0,C 180,E1 -26965.763,E2 -26965.763} C_VEL
LIN {X 0,Y 116.048,Z 360.472,A -85,B 0,C 180,E1 -26969.017,E2 -26969.017} C_VEL
LIN {X 0,Y 113.159,Z 356.374,A -85,B 0,C 180,E1 -26972.863,E2 -26972.863} C_VEL
LIN {X 0,Y 110.697,Z 353.361,A -85,B 0,C 180,E1 -26976.832,E2 -26976.832} C_VEL
LIN {X 0,Y 109.713,Z 351.519,A -85,B 0,C 180,E1 -26978.879,E2 -26978.879} C_VEL
LIN {X 0,Y 106.985,Z 348.883,A -85,B 0,C 180,E1 -26986.113,E2 -26986.113} C_VEL
LIN {X 0,Y 106.235,Z 346.035,A -85,B 0,C 180,E1 -26991.435,E2 -26991.435} C_VEL
LIN {X 0,Y 106.455,Z 346.057,A -85,B 0,C 180,E1 -27000.472,E2 -27000.472} C_VEL
LIN {X 0,Y 107.27,Z 348.868,A -85,B 0,C 180,E1 -27005.168,E2 -27005.168} C_VEL
LIN {X 0,Y 110.085,Z 351.84,A -85,B 0,C 180,E1 -27012.208,E2 -27012.208} C_VEL
LIN {X 0,Y 111.945,Z 355.141,A -85,B 0,C 180,E1 -27015.708,E2 -27015.708} C_VEL
LIN {X 0,Y 113.64,Z 356.949,A -85,B 0,C 180,E1 -27018.186,E2 -27018.186} C_VEL
LIN {X 0,Y 116.185,Z 360.649,A -85,B 0,C 180,E1 -27021.513,E2 -27021.513} C_VEL
LIN {X 0,Y 119.855,Z 366.123,A -85,B 0,C 180,E1 -27025.535,E2 -27025.535} C_VEL
LIN {X 0,Y 123.833,Z 372.677,A -85,B 0,C 180,E1 -27029.249,E2 -27029.249} C_VEL
LIN {X 0,Y 125.807,Z 376.782,A -85,B 0,C 180,E1 -27030.967,E2 -27030.967} C_VEL
LIN {X 0,Y 129.428,Z 386.639,A -85,B 0,C 180,E1 -27034.024,E2 -27034.024} C_VEL
LIN {X 0,Y 131.235,Z 392.563,A -85,B 0,C 180,E1 -27035.5,E2 -27035.5} C_VEL
LIN {X 0,Y 131.359,Z 400.658,A -85,B 0,C 180,E1 -27036.235,E2 -27036.235} C_VEL
LIN {X 0,Y 128.413,Z 435.351,A -85,B 0,C 180,E1 -27037.784,E2 -27037.784} C_VEL
LIN {X 0,Y 126.302,Z 448.344,A -85,B 0,C 180,E1 -27038.826,E2 -27038.826} C_VEL
LIN {X 0,Y 123.276,Z 460.855,A -85,B 0,C 180,E1 -27040.311,E2 -27040.311} C_VEL
LIN {X 0,Y 119.637,Z 471.973,A -85,B 0,C 180,E1 -27042.125,E2 -27042.125} C_VEL
LIN {X 0,Y 115.19,Z 483.608,A -85,B 0,C 180,E1 -27044.822,E2 -27044.822} C_VEL
LIN {X 0,Y 110.972,Z 492.989,A -85,B 0,C 180,E1 -27047.706,E2 -27047.706} C_VEL
LIN {X 0,Y 106.607,Z 501.715,A -85,B 0,C 180,E1 -27051.221,E2 -27051.221} C_VEL
LIN {X 0,Y 102.04,Z 510.21,A -85,B 0,C 180,E1 -27055.74,E2 -27055.74} C_VEL
LIN {X 0,Y 98.111,Z 517.621,A -85,B 0,C 180,E1 -27061.081,E2 -27061.081} C_VEL
LIN {X 0,Y 95.324,Z 522.981,A -85,B 0,C 180,E1 -27066.075,E2 -27066.075} C_VEL
LIN {X 0,Y 92.828,Z 528.167,A -85,B 0,C 180,E1 -27072.369,E2 -27072.369} C_VEL
LIN {X 0,Y 91.504,Z 532.189,A -85,B 0,C 180,E1 -27078.927,E2 -27078.927} C_VEL
LIN {X 0,Y 91.12,Z 535.143,A -85,B 0,C 180,E1 -27085.574,E2 -27085.574} C_VEL
LIN {X 0,Y 91.329,Z 536.538,A -85,B 0,C 180,E1 -27089.997,E2 -27089.997} C_VEL
LIN {X 0,Y 91.076,Z 537.476,A -85,B 0,C 180,E1 -27094.423,E2 -27094.423} C_VEL
LIN {X 0,Y 91.257,Z 538.028,A -85,B 0,C 180,E1 -27098.858,E2 -27098.858} C_VEL
LIN {X 0,Y 91.832,Z 538.192,A -85,B 0,C 180,E1 -27103.27,E2 -27103.27} C_VEL
LIN {X 0,Y 94.52,Z 537.291,A -85,B 0,C 180,E1 -27111.822,E2 -27111.822} C_VEL
LIN {X 0,Y 99.32,Z 534.865,A -85,B 0,C 180,E1 -27119.688,E2 -27119.688} C_VEL
LIN {X 0,Y 104.05,Z 531.931,A -85,B 0,C 180,E1 -27125.035,E2 -27125.035} C_VEL
LIN {X 0,Y 109.522,Z 527.989,A -85,B 0,C 180,E1 -27129.915,E2 -27129.915} C_VEL
LIN {X 0,Y 115.733,Z 522.942,A -85,B 0,C 180,E1 -27134.292,E2 -27134.292} C_VEL
LIN {X 0,Y 122.686,Z 516.637,A -85,B 0,C 180,E1 -27138.13,E2 -27138.13} C_VEL
LIN {X 0,Y 130.189,Z 508.772,A -85,B 0,C 180,E1 -27141.51,E2 -27141.51} C_VEL
LIN {X 0,Y 138.069,Z 499.001,A -85,B 0,C 180,E1 -27144.528,E2 -27144.528} C_VEL
LIN {X 0,Y 145.04,Z 488.867,A -85,B 0,C 180,E1 -27146.702,E2 -27146.702} C_VEL
LIN {X 0,Y 150.75,Z 478.843,A -85,B 0,C 180,E1 -27148.298,E2 -27148.298} C_VEL
LIN {X 0,Y 155.857,Z 467.948,A -85,B 0,C 180,E1 -27149.583,E2 -27149.583} C_VEL
LIN {X 0,Y 160.296,Z 455.924,A -85,B 0,C 180,E1 -27150.618,E2 -27150.618} C_VEL
LIN {X 0,Y 163.647,Z 443.521,A -85,B 0,C 180,E1 -27151.383,E2 -27151.383} C_VEL
LIN {X 0,Y 165.958,Z 429.668,A -85,B 0,C 180,E1 -27151.954,E2 -27151.954} C_VEL
LIN {X 0,Y 166.503,Z 424.058,A -85,B 0,C 180,E1 -27152.165,E2 -27152.165} C_VEL
LIN {X 0,Y 164.15,Z 416.642,A -85,B 0,C 180,E1 -27154.959,E2 -27154.959} C_VEL
LIN {X 0,Y 163.809,Z 415.641,A -85,B 0,C 180,E1 -27155.392,E2 -27155.392} C_VEL
LIN {X 0,Y 162.926,Z 413.519,A -85,B 0,C 180,E1 -27156.505,E2 -27156.505} C_VEL
LIN {X 0,Y 161.392,Z 411.504,A -85,B 0,C 180,E1 -27158.395,E2 -27158.395} C_VEL
LIN {X 0,Y 158.857,Z 409.942,A -85,B 0,C 180,E1 -27161.844,E2 -27161.844} C_VEL
LIN {X 0,Y 156.912,Z 408.253,A -85,B 0,C 180,E1 -27165.438,E2 -27165.438} C_VEL
LIN {X 0,Y 156.643,Z 407.647,A -85,B 0,C 180,E1 -27166.144,E2 -27166.144} C_VEL
LIN {X 0,Y 156.129,Z 406.527,A -85,B 0,C 180,E1 -27167.654,E2 -27167.654} C_VEL
LIN {X 0,Y 154.978,Z 403.432,A -85,B 0,C 180,E1 -27173.983,E2 -27173.983} C_VEL
LIN {X 0,Y 154.981,Z 402.93,A -85,B 0,C 180,E1 -27174.797,E2 -27174.797} C_VEL
LIN {X 0,Y 155.009,Z 402.959,A -85,B 0,C 180,E1 -27177.402,E2 -27177.402} C_VEL
LIN {X 0,Y 155.652,Z 405.561,A -85,B 0,C 180,E1 -27182.346,E2 -27182.346} C_VEL
LIN {X 0,Y 156.46,Z 406.84,A -85,B 0,C 180,E1 -27184.913,E2 -27184.913} C_VEL
LIN {X 0,Y 158.346,Z 410.873,A -85,B 0,C 180,E1 -27189.259,E2 -27189.259} C_VEL
LIN {X 0,Y 160.223,Z 414.773,A -85,B 0,C 180,E1 -27192.428,E2 -27192.428} C_VEL
LIN {X 0,Y 162.717,Z 420.15,A -85,B 0,C 180,E1 -27195.823,E2 -27195.823} C_VEL
LIN {X 0,Y 163.825,Z 422.872,A -85,B 0,C 180,E1 -27197.205,E2 -27197.205} C_VEL
LIN {X 0,Y 161.801,Z 435.693,A -85,B 0,C 180,E1 -27197.761,E2 -27197.761} C_VEL
LIN {X 0,Y 158.959,Z 447.14,A -85,B 0,C 180,E1 -27198.491,E2 -27198.491} C_VEL
LIN {X 0,Y 154.728,Z 459.369,A -85,B 0,C 180,E1 -27199.529,E2 -27199.529} C_VEL
LIN {X 0,Y 149.46,Z 470.872,A -85,B 0,C 180,E1 -27200.845,E2 -27200.845} C_VEL
LIN {X 0,Y 143.011,Z 482.368,A -85,B 0,C 180,E1 -27202.747,E2 -27202.747} C_VEL
LIN {X 0,Y 137.311,Z 490.898,A -85,B 0,C 180,E1 -27204.706,E2 -27204.706} C_VEL
LIN {X 0,Y 130.425,Z 499.558,A -85,B 0,C 180,E1 -27207.243,E2 -27207.243} C_VEL
LIN {X 0,Y 122.478,Z 507.915,A -85,B 0,C 180,E1 -27210.606,E2 -27210.606} C_VEL
LIN {X 0,Y 115.051,Z 514.611,A -85,B 0,C 180,E1 -27214.45,E2 -27214.45} C_VEL
LIN {X 0,Y 108.111,Z 519.914,A -85,B 0,C 180,E1 -27218.735,E2 -27218.735} C_VEL
LIN {X 0,Y 101.537,Z 524.188,A -85,B 0,C 180,E1 -27223.803,E2 -27223.803} C_VEL
LIN {X 0,Y 96.313,Z 527.016,A -85,B 0,C 180,E1 -27228.952,E2 -27228.952} C_VEL
LIN {X 0,Y 93.145,Z 528.473,A -85,B 0,C 180,E1 -27232.874,E2 -27232.874} C_VEL
LIN {X 0,Y 88.173,Z 530.083,A -85,B 0,C 180,E1 -27241.433,E2 -27241.433} C_VEL
LIN {X 0,Y 86.364,Z 530.303,A -85,B 0,C 180,E1 -27245.994,E2 -27245.994} C_VEL
LIN {X 0,Y 85.007,Z 530.101,A -85,B 0,C 180,E1 -27250.692,E2 -27250.692} C_VEL
LIN {X 0,Y 83.931,Z 528.471,A -85,B 0,C 180,E1 -27260.362,E2 -27260.362} C_VEL
LIN {X 0,Y 84.426,Z 526.26,A -85,B 0,C 180,E1 -27267.389,E2 -27267.389} C_VEL
LIN {X 0,Y 85.6,Z 522.933,A -85,B 0,C 180,E1 -27274.712,E2 -27274.712} C_VEL
LIN {X 0,Y 87.788,Z 518.636,A -85,B 0,C 180,E1 -27281.548,E2 -27281.548} C_VEL
LIN {X 0,Y 91.632,Z 512.146,A -85,B 0,C 180,E1 -27289.027,E2 -27289.027} C_VEL
LIN {X 0,Y 95.887,Z 505.028,A -85,B 0,C 180,E1 -27294.929,E2 -27294.929} C_VEL
LIN {X 0,Y 101.016,Z 496.174,A -85,B 0,C 180,E1 -27300.295,E2 -27300.295} C_VEL
LIN {X 0,Y 105.934,Z 487.078,A -85,B 0,C 180,E1 -27304.33,E2 -27304.33} C_VEL
LIN {X 0,Y 110.716,Z 476.988,A -85,B 0,C 180,E1 -27307.663,E2 -27307.663} C_VEL
LIN {X 0,Y 115.161,Z 465.803,A -85,B 0,C 180,E1 -27310.425,E2 -27310.425} C_VEL
LIN {X 0,Y 119.079,Z 453.292,A -85,B 0,C 180,E1 -27312.747,E2 -27312.747} C_VEL
LIN {X 0,Y 122.207,Z 440.23,A -85,B 0,C 180,E1 -27314.373,E2 -27314.373} C_VEL
LIN {X 0,Y 124.307,Z 427.162,A -85,B 0,C 180,E1 -27315.451,E2 -27315.451} C_VEL
LIN {X 0,Y 127.344,Z 391.68,A -85,B 0,C 180,E1 -27317.07,E2 -27317.07} C_VEL
LIN {X 0,Y 123.824,Z 383.924,A -85,B 0,C 180,E1 -27319.982,E2 -27319.982} C_VEL
LIN {X 0,Y 120.03,Z 376.75,A -85,B 0,C 180,E1 -27323.464,E2 -27323.464} C_VEL
LIN {X 0,Y 116.174,Z 370.248,A -85,B 0,C 180,E1 -27327.571,E2 -27327.571} C_VEL
LIN {X 0,Y 113.799,Z 366.547,A -85,B 0,C 180,E1 -27330.518,E2 -27330.518} C_VEL
LIN {X 0,Y 111.38,Z 362.903,A -85,B 0,C 180,E1 -27334.038,E2 -27334.038} C_VEL
LIN {X 0,Y 108.89,Z 359.461,A -85,B 0,C 180,E1 -27338.525,E2 -27338.525} C_VEL
LIN {X 0,Y 108.38,Z 358.365,A -85,B 0,C 180,E1 -27339.724,E2 -27339.724} C_VEL
LIN {X 0,Y 105.8,Z 355.512,A -85,B 0,C 180,E1 -27347.429,E2 -27347.429} C_VEL
LIN {X 0,Y 105.321,Z 353.061,A -85,B 0,C 180,E1 -27351.845,E2 -27351.845} C_VEL
LIN {X 0,Y 105.463,Z 352.941,A -85,B 0,C 180,E1 -27359.569,E2 -27359.569} C_VEL
LIN {X 0,Y 106.197,Z 355.784,A -85,B 0,C 180,E1 -27364.506,E2 -27364.506} C_VEL
LIN {X 0,Y 108.59,Z 358.526,A -85,B 0,C 180,E1 -27371.077,E2 -27371.077} C_VEL
LIN {X 0,Y 110.398,Z 361.817,A -85,B 0,C 180,E1 -27374.751,E2 -27374.751} C_VEL
LIN {X 0,Y 111.822,Z 363.516,A -85,B 0,C 180,E1 -27377.016,E2 -27377.016} C_VEL
LIN {X 0,Y 115.003,Z 368.386,A -85,B 0,C 180,E1 -27381.392,E2 -27381.392} C_VEL
LIN {X 0,Y 117.636,Z 372.568,A -85,B 0,C 180,E1 -27384.426,E2 -27384.426} C_VEL
LIN {X 0,Y 121.473,Z 379.352,A -85,B 0,C 180,E1 -27388.274,E2 -27388.274} C_VEL
LIN {X 0,Y 124.934,Z 388.996,A -85,B 0,C 180,E1 -27391.591,E2 -27391.591} C_VEL
LIN {X 0,Y 126.793,Z 395.333,A -85,B 0,C 180,E1 -27393.304,E2 -27393.304} C_VEL
LIN {X 0,Y 126.716,Z 402.316,A -85,B 0,C 180,E1 -27393.89,E2 -27393.89} C_VEL
LIN {X 0,Y 123.762,Z 435.07,A -85,B 0,C 180,E1 -27395.344,E2 -27395.344} C_VEL
LIN {X 0,Y 121.478,Z 448.484,A -85,B 0,C 180,E1 -27396.431,E2 -27396.431} C_VEL
LIN {X 0,Y 118.153,Z 461.34,A -85,B 0,C 180,E1 -27397.985,E2 -27397.985} C_VEL
LIN {X 0,Y 113.801,Z 473.892,A -85,B 0,C 180,E1 -27400.157,E2 -27400.157} C_VEL
LIN {X 0,Y 109.111,Z 485.097,A -85,B 0,C 180,E1 -27402.885,E2 -27402.885} C_VEL
LIN {X 0,Y 104.207,Z 495.163,A -85,B 0,C 180,E1 -27406.264,E2 -27406.264} C_VEL
LIN {X 0,Y 99.264,Z 504.289,A -85,B 0,C 180,E1 -27410.413,E2 -27410.413} C_VEL
LIN {X 0,Y 94.554,Z 512.072,A -85,B 0,C 180,E1 -27415.086,E2 -27415.086} C_VEL
LIN {X 0,Y 91.932,Z 516.953,A -85,B 0,C 180,E1 -27418.931,E2 -27418.931} C_VEL
LIN {X 0,Y 88.857,Z 522.353,A -85,B 0,C 180,E1 -27424.211,E2 -27424.211} C_VEL
LIN {X 0,Y 86.042,Z 527.608,A -85,B 0,C 180,E1 -27430.927,E2 -27430.927} C_VEL
LIN {X 0,Y 84.507,Z 531.686,A -85,B 0,C 180,E1 -27437.997,E2 -27437.997} C_VEL
LIN {X 0,Y 84.044,Z 534.686,A -85,B 0,C 180,E1 -27445.2,E2 -27445.2} C_VEL
LIN {X 0,Y 84.247,Z 536.124,A -85,B 0,C 180,E1 -27449.997,E2 -27449.997} C_VEL
LIN {X 0,Y 84.232,Z 537.661,A -85,B 0,C 180,E1 -27459.603,E2 -27459.603} C_VEL
LIN {X 0,Y 84.92,Z 537.851,A -85,B 0,C 180,E1 -27464.373,E2 -27464.373} C_VEL
LIN {X 0,Y 86.172,Z 537.64,A -85,B 0,C 180,E1 -27469.037,E2 -27469.037} C_VEL
LIN {X 0,Y 90.325,Z 536.024,A -85,B 0,C 180,E1 -27477.827,E2 -27477.827} C_VEL
LIN {X 0,Y 93.186,Z 534.642,A -85,B 0,C 180,E1 -27481.863,E2 -27481.863} C_VEL
LIN {X 0,Y 98.292,Z 531.758,A -85,B 0,C 180,E1 -27487.424,E2 -27487.424} C_VEL
LIN {X 0,Y 104.162,Z 527.87,A -85,B 0,C 180,E1 -27492.429,E2 -27492.429} C_VEL
LIN {X 0,Y 110.759,Z 522.881,A -85,B 0,C 180,E1 -27496.859,E2 -27496.859} C_VEL
LIN {X 0,Y 118.065,Z 516.641,A -85,B 0,C 180,E1 -27500.697,E2 -27500.697} C_VEL
LIN {X 0,Y 125.89,Z 508.884,A -85,B 0,C 180,E1 -27504.042,E2 -27504.042} C_VEL
LIN {X 0,Y 134.089,Z 499.201,A -85,B 0,C 180,E1 -27506.99,E2 -27506.99} C_VEL
LIN {X 0,Y 141.275,Z 489.216,A -85,B 0,C 180,E1 -27509.104,E2 -27509.104} C_VEL
LIN {X 0,Y 147.163,Z 479.361,A -85,B 0,C 180,E1 -27510.637,E2 -27510.637} C_VEL
LIN {X 0,Y 152.406,Z 468.669,A -85,B 0,C 180,E1 -27511.872,E2 -27511.872} C_VEL
LIN {X 0,Y 157.335,Z 455.813,A -85,B 0,C 180,E1 -27512.943,E2 -27512.943} C_VEL
LIN {X 0,Y 160.873,Z 443.116,A -85,B 0,C 180,E1 -27513.683,E2 -27513.683} C_VEL
LIN {X 0,Y 163.165,Z 429.763,A -85,B 0,C 180,E1 -27514.227,E2 -27514.227} C_VEL
LIN {X 0,Y 163.432,Z 427.099,A -85,B 0,C 180,E1 -27514.361,E2 -27514.361} C_VEL
LIN {X 0,Y 161.014,Z 419.074,A -85,B 0,C 180,E1 -27517.726,E2 -27517.726} C_VEL
LIN {X 0,Y 158.895,Z 412.675,A -85,B 0,C 180,E1 -27521.297,E2 -27521.297} C_VEL
LIN {X 0,Y 157.785,Z 409.863,A -85,B 0,C 180,E1 -27523.504,E2 -27523.504} C_VEL
LIN {X 0,Y 156.643,Z 407.647,A -85,B 0,C 180,E1 -27526.144,E2 -27526.144} C_VEL
LIN {X 0,Y 155.91,Z 406.478,A -85,B 0,C 180,E1 -27528.244,E2 -27528.244} C_VEL
LIN {X 0,Y 155.221,Z 406.544,A -85,B 0,C 180,E1 -27530.416,E2 -27530.416} C_VEL
LIN {X 0,Y 154.501,Z 407.847,A -85,B 0,C 180,E1 -27533.345,E2 -27533.345} C_VEL
LIN {X 0,Y 154.12,Z 410.437,A -85,B 0,C 180,E1 -27537.792,E2 -27537.792} C_VEL
LIN {X 0,Y 155.359,Z 413.703,A -85,B 0,C 180,E1 -27544.338,E2 -27544.338} C_VEL
LIN {X 0,Y 157.132,Z 417.797,A -85,B 0,C 180,E1 -27548.739,E2 -27548.739} C_VEL
LIN {X 0,Y 159.27,Z 422.557,A -85,B 0,C 180,E1 -27552.504,E2 -27552.504} C_VEL
LIN {X 0,Y 160.876,Z 426.682,A -85,B 0,C 180,E1 -27554.978,E2 -27554.978} C_VEL
LIN {X 0,Y 158.36,Z 439.897,A -85,B 0,C 180,E1 -27555.625,E2 -27555.625} C_VEL
LIN {X 0,Y 154.765,Z 452.277,A -85,B 0,C 180,E1 -27556.484,E2 -27556.484} C_VEL
LIN {X 0,Y 150.158,Z 463.89,A -85,B 0,C 180,E1 -27557.521,E2 -27557.521} C_VEL
LIN {X 0,Y 144.791,Z 474.543,A -85,B 0,C 180,E1 -27558.83,E2 -27558.83} C_VEL
LIN {X 0,Y 138.91,Z 484.184,A -85,B 0,C 180,E1 -27560.462,E2 -27560.462} C_VEL
LIN {X 0,Y 131.565,Z 494.292,A -85,B 0,C 180,E1 -27562.863,E2 -27562.863} C_VEL
LIN {X 0,Y 124.464,Z 502.393,A -85,B 0,C 180,E1 -27565.388,E2 -27565.388} C_VEL
LIN {X 0,Y 116.624,Z 509.99,A -85,B 0,C 180,E1 -27568.643,E2 -27568.643} C_VEL
LIN {X 0,Y 108.575,Z 516.545,A -85,B 0,C 180,E1 -27572.708,E2 -27572.708} C_VEL
LIN {X 0,Y 101.405,Z 521.487,A -85,B 0,C 180,E1 -27577.157,E2 -27577.157} C_VEL
LIN {X 0,Y 94.874,Z 525.269,A -85,B 0,C 180,E1 -27582.207,E2 -27582.207} C_VEL
LIN {X 0,Y 90.968,Z 527.202,A -85,B 0,C 180,E1 -27585.951,E2 -27585.951} C_VEL
LIN {X 0,Y 87.471,Z 528.707,A -85,B 0,C 180,E1 -27590.005,E2 -27590.005} C_VEL
LIN {X 0,Y 84.433,Z 529.745,A -85,B 0,C 180,E1 -27594.366,E2 -27594.366} C_VEL
LIN {X 0,Y 79.805,Z 530.626,A -85,B 0,C 180,E1 -27603.879,E2 -27603.879} C_VEL
LIN {X 0,Y 78.247,Z 530.474,A -85,B 0,C 180,E1 -27608.948,E2 -27608.948} C_VEL
LIN {X 0,Y 77.269,Z 529.882,A -85,B 0,C 180,E1 -27614.169,E2 -27614.169} C_VEL
LIN {X 0,Y 76.856,Z 528.9,A -85,B 0,C 180,E1 -27619.465,E2 -27619.465} C_VEL
LIN {X 0,Y 77.368,Z 526.523,A -85,B 0,C 180,E1 -27627.778,E2 -27627.778} C_VEL
LIN {X 0,Y 78.539,Z 523.468,A -85,B 0,C 180,E1 -27635.137,E2 -27635.137} C_VEL
LIN {X 0,Y 80.832,Z 519.235,A -85,B 0,C 180,E1 -27642.557,E2 -27642.557} C_VEL
LIN {X 0,Y 84.963,Z 512.817,A -85,B 0,C 180,E1 -27650.586,E2 -27650.586} C_VEL
LIN {X 0,Y 89.524,Z 505.805,A -85,B 0,C 180,E1 -27656.837,E2 -27656.837} C_VEL
LIN {X 0,Y 94.968,Z 497.043,A -85,B 0,C 180,E1 -27662.451,E2 -27662.451} C_VEL
LIN {X 0,Y 100.724,Z 487.072,A -85,B 0,C 180,E1 -27667.002,E2 -27667.002} C_VEL
LIN {X 0,Y 105.801,Z 476.882,A -85,B 0,C 180,E1 -27670.369,E2 -27670.369} C_VEL
LIN {X 0,Y 110.482,Z 465.604,A -85,B 0,C 180,E1 -27673.147,E2 -27673.147} C_VEL
LIN {X 0,Y 114.312,Z 453.949,A -85,B 0,C 180,E1 -27675.309,E2 -27675.309} C_VEL
LIN {X 0,Y 117.492,Z 441.54,A -85,B 0,C 180,E1 -27676.881,E2 -27676.881} C_VEL
LIN {X 0,Y 119.795,Z 428.315,A -85,B 0,C 180,E1 -27677.989,E2 -27677.989} C_VEL
LIN {X 0,Y 122.168,Z 403.31,A -85,B 0,C 180,E1 -27679.145,E2 -27679.145} C_VEL
LIN {X 0,Y 122.898,Z 394.357,A -85,B 0,C 180,E1 -27679.555,E2 -27679.555} C_VEL
LIN {X 0,Y 119.76,Z 387.337,A -85,B 0,C 180,E1 -27682.492,E2 -27682.492} C_VEL
LIN {X 0,Y 116.677,Z 381.358,A -85,B 0,C 180,E1 -27685.69,E2 -27685.69} C_VEL
LIN {X 0,Y 113.493,Z 375.724,A -85,B 0,C 180,E1 -27689.5,E2 -27689.5} C_VEL
LIN {X 0,Y 111.693,Z 372.733,A -85,B 0,C 180,E1 -27691.983,E2 -27691.983} C_VEL
LIN {X 0,Y 109.582,Z 369.355,A -85,B 0,C 180,E1 -27695.361,E2 -27695.361} C_VEL
LIN {X 0,Y 107.154,Z 365.45,A -85,B 0,C 180,E1 -27700.357,E2 -27700.357} C_VEL
LIN {X 0,Y 104.599,Z 361.821,A -85,B 0,C 180,E1 -27709.351,E2 -27709.351} C_VEL
LIN {X 0,Y 104.402,Z 360.165,A -85,B 0,C 180,E1 -27712.262,E2 -27712.262} C_VEL
LIN {X 0,Y 104.504,Z 360.092,A -85,B 0,C 180,E1 -27718.997,E2 -27718.997} C_VEL
LIN {X 0,Y 105.614,Z 363.567,A -85,B 0,C 180,E1 -27725.728,E2 -27725.728} C_VEL
LIN {X 0,Y 107.181,Z 365.309,A -85,B 0,C 180,E1 -27730.026,E2 -27730.026} C_VEL
LIN {X 0,Y 109.18,Z 368.821,A -85,B 0,C 180,E1 -27734.297,E2 -27734.297} C_VEL
LIN {X 0,Y 110.15,Z 370.231,A -85,B 0,C 180,E1 -27735.97,E2 -27735.97} C_VEL
LIN {X 0,Y 112.951,Z 374.769,A -85,B 0,C 180,E1 -27740.145,E2 -27740.145} C_VEL
LIN {X 0,Y 115.994,Z 379.911,A -85,B 0,C 180,E1 -27743.881,E2 -27743.881} C_VEL
LIN {X 0,Y 118.644,Z 385.257,A -85,B 0,C 180,E1 -27746.776,E2 -27746.776} C_VEL
LIN {X 0,Y 121.742,Z 394.854,A -85,B 0,C 180,E1 -27750.085,E2 -27750.085} C_VEL
LIN {X 0,Y 122.518,Z 397.814,A -85,B 0,C 180,E1 -27750.902,E2 -27750.902} C_VEL
LIN {X 0,Y 122.307,Z 403.737,A -85,B 0,C 180,E1 -27751.351,E2 -27751.351} C_VEL
LIN {X 0,Y 119.412,Z 434.362,A -85,B 0,C 180,E1 -27752.69,E2 -27752.69} C_VEL
LIN {X 0,Y 117.224,Z 447.092,A -85,B 0,C 180,E1 -27753.706,E2 -27753.706} C_VEL
LIN {X 0,Y 113.882,Z 459.766,A -85,B 0,C 180,E1 -27755.141,E2 -27755.141} C_VEL
LIN {X 0,Y 109.941,Z 471.005,A -85,B 0,C 180,E1 -27756.955,E2 -27756.955} C_VEL
LIN {X 0,Y 104.968,Z 482.686,A -85,B 0,C 180,E1 -27759.646,E2 -27759.646} C_VEL
LIN {X 0,Y 99.725,Z 493.2,A -85,B 0,C 180,E1 -27763.012,E2 -27763.012} C_VEL
LIN {X 0,Y 94.837,Z 501.78,A -85,B 0,C 180,E1 -27766.723,E2 -27766.723} C_VEL
LIN {X 0,Y 89.666,Z 510.119,A -85,B 0,C 180,E1 -27771.608,E2 -27771.608} C_VEL
LIN {X 0,Y 87.491,Z 513.619,A -85,B 0,C 180,E1 -27774.217,E2 -27774.217} C_VEL
LIN {X 0,Y 83.1,Z 520.694,A -85,B 0,C 180,E1 -27780.899,E2 -27780.899} C_VEL
LIN {X 0,Y 79.303,Z 527.035,A -85,B 0,C 180,E1 -27789.235,E2 -27789.235} C_VEL
LIN {X 0,Y 77.552,Z 531.171,A -85,B 0,C 180,E1 -27796.902,E2 -27796.902} C_VEL
LIN {X 0,Y 76.965,Z 534.222,A -85,B 0,C 180,E1 -27804.757,E2 -27804.757} C_VEL
LIN {X 0,Y 77.154,Z 535.71,A -85,B 0,C 180,E1 -27809.997,E2 -27809.997} C_VEL
LIN {X 0,Y 77.219,Z 537.293,A -85,B 0,C 180,E1 -27820.485,E2 -27820.485} C_VEL
LIN {X 0,Y 79.46,Z 537.338,A -85,B 0,C 180,E1 -27830.716,E2 -27830.716} C_VEL
LIN {X 0,Y 84.088,Z 535.776,A -85,B 0,C 180,E1 -27840.094,E2 -27840.094} C_VEL
LIN {X 0,Y 90.816,Z 532.661,A -85,B 0,C 180,E1 -27848.247,E2 -27848.247} C_VEL
LIN {X 0,Y 95.855,Z 529.733,A -85,B 0,C 180,E1 -27852.847,E2 -27852.847} C_VEL
LIN {X 0,Y 103.596,Z 524.616,A -85,B 0,C 180,E1 -27858.262,E2 -27858.262} C_VEL
LIN {X 0,Y 112.368,Z 517.764,A -85,B 0,C 180,E1 -27862.882,E2 -27862.882} C_VEL
LIN {X 0,Y 120.491,Z 510.356,A -85,B 0,C 180,E1 -27866.216,E2 -27866.216} C_VEL
LIN {X 0,Y 127.506,Z 502.832,A -85,B 0,C 180,E1 -27868.683,E2 -27868.683} C_VEL
LIN {X 0,Y 134.774,Z 493.743,A -85,B 0,C 180,E1 -27870.859,E2 -27870.859} C_VEL
LIN {X 0,Y 141.561,Z 483.703,A -85,B 0,C 180,E1 -27872.548,E2 -27872.548} C_VEL
LIN {X 0,Y 147.645,Z 472.572,A -85,B 0,C 180,E1 -27873.953,E2 -27873.953} C_VEL
LIN {X 0,Y 153.094,Z 460.09,A -85,B 0,C 180,E1 -27875.043,E2 -27875.043} C_VEL
LIN {X 0,Y 157.126,Z 447.521,A -85,B 0,C 180,E1 -27875.846,E2 -27875.846} C_VEL
LIN {X 0,Y 160.035,Z 433.981,A -85,B 0,C 180,E1 -27876.437,E2 -27876.437} C_VEL
LIN {X 0,Y 160.523,Z 430.276,A -85,B 0,C 180,E1 -27876.624,E2 -27876.624} C_VEL
LIN {X 0,Y 158.693,Z 423.55,A -85,B 0,C 180,E1 -27879.738,E2 -27879.738} C_VEL
LIN {X 0,Y 157.242,Z 418.598,A -85,B 0,C 180,E1 -27882.609,E2 -27882.609} C_VEL
LIN {X 0,Y 156.378,Z 416.347,A -85,B 0,C 180,E1 -27884.524,E2 -27884.524} C_VEL
LIN {X 0,Y 155.055,Z 413.388,A -85,B 0,C 180,E1 -27888.232,E2 -27888.232} C_VEL
LIN {X 0,Y 154.087,Z 410.189,A -85,B 0,C 180,E1 -27894.767,E2 -27894.767} C_VEL
LIN {X 0,Y 154.116,Z 410.386,A -85,B 0,C 180,E1 -27897.681,E2 -27897.681} C_VEL
LIN {X 0,Y 154.12,Z 410.437,A -85,B 0,C 180,E1 -27897.792,E2 -27897.792} C_VEL
LIN {X 0,Y 154.229,Z 412.074,A -85,B 0,C 180,E1 -27899.902,E2 -27899.902} C_VEL
LIN {X 0,Y 154.4,Z 414.648,A -85,B 0,C 180,E1 -27901.89,E2 -27901.89} C_VEL
LIN {X 0,Y 155.045,Z 420.966,A -85,B 0,C 180,E1 -27905.676,E2 -27905.676} C_VEL
LIN {X 0,Y 155.898,Z 424.798,A -85,B 0,C 180,E1 -27908.261,E2 -27908.261} C_VEL
LIN {X 0,Y 157.43,Z 428.834,A -85,B 0,C 180,E1 -27911.485,E2 -27911.485} C_VEL
LIN {X 0,Y 158.02,Z 430.654,A -85,B 0,C 180,E1 -27912.686,E2 -27912.686} C_VEL
LIN {X 0,Y 155.459,Z 442.474,A -85,B 0,C 180,E1 -27913.291,E2 -27913.291} C_VEL
LIN {X 0,Y 151.738,Z 454.385,A -85,B 0,C 180,E1 -27914.135,E2 -27914.135} C_VEL
LIN {X 0,Y 146.555,Z 466.422,A -85,B 0,C 180,E1 -27915.191,E2 -27915.191} C_VEL
LIN {X 0,Y 141.068,Z 476.629,A -85,B 0,C 180,E1 -27916.463,E2 -27916.463} C_VEL
LIN {X 0,Y 134.761,Z 486.344,A -85,B 0,C 180,E1 -27918.119,E2 -27918.119} C_VEL
LIN {X 0,Y 127.426,Z 495.825,A -85,B 0,C 180,E1 -27920.351,E2 -27920.351} C_VEL
LIN {X 0,Y 120.087,Z 503.715,A -85,B 0,C 180,E1 -27922.822,E2 -27922.822} C_VEL
LIN {X 0,Y 111.632,Z 511.329,A -85,B 0,C 180,E1 -27926.15,E2 -27926.15} C_VEL
LIN {X 0,Y 102.229,Z 518.392,A -85,B 0,C 180,E1 -27930.762,E2 -27930.762} C_VEL
LIN {X 0,Y 94.774,Z 523.006,A -85,B 0,C 180,E1 -27935.347,E2 -27935.347} C_VEL
LIN {X 0,Y 90.161,Z 525.426,A -85,B 0,C 180,E1 -27938.79,E2 -27938.79} C_VEL
LIN {X 0,Y 85.902,Z 527.387,A -85,B 0,C 180,E1 -27942.585,E2 -27942.585} C_VEL
LIN {X 0,Y 82.038,Z 528.925,A -85,B 0,C 180,E1 -27946.742,E2 -27946.742} C_VEL
LIN {X 0,Y 78.656,Z 530.014,A -85,B 0,C 180,E1 -27951.288,E2 -27951.288} C_VEL
LIN {X 0,Y 73.379,Z 530.948,A -85,B 0,C 180,E1 -27961.392,E2 -27961.392} C_VEL
LIN {X 0,Y 71.576,Z 530.833,A -85,B 0,C 180,E1 -27966.878,E2 -27966.878} C_VEL
LIN {X 0,Y 70.372,Z 530.285,A -85,B 0,C 180,E1 -27972.57,E2 -27972.57} C_VEL
LIN {X 0,Y 69.876,Z 527.978,A -85,B 0,C 180,E1 -27984.231,E2 -27984.231} C_VEL
LIN {X 0,Y 70.907,Z 525.158,A -85,B 0,C 180,E1 -27992.844,E2 -27992.844} C_VEL
LIN {X 0,Y 72.918,Z 521.348,A -85,B 0,C 180,E1 -28001.118,E2 -28001.118} C_VEL
LIN {X 0,Y 76.319,Z 516.406,A -85,B 0,C 180,E1 -28008.806,E2 -28008.806} C_VEL
LIN {X 0,Y 80.722,Z 510.211,A -85,B 0,C 180,E1 -28015.809,E2 -28015.809} C_VEL
LIN {X 0,Y 86.06,Z 502.484,A -85,B 0,C 180,E1 -28022.064,E2 -28022.064} C_VEL
LIN {X 0,Y 92.319,Z 492.801,A -85,B 0,C 180,E1 -28027.522,E2 -28027.522} C_VEL
LIN {X 0,Y 98.12,Z 482.771,A -85,B 0,C 180,E1 -28031.498,E2 -28031.498} C_VEL
LIN {X 0,Y 103.622,Z 471.411,A -85,B 0,C 180,E1 -28034.725,E2 -28034.725} C_VEL
LIN {X 0,Y 107.945,Z 460.318,A -85,B 0,C 180,E1 -28037.096,E2 -28037.096} C_VEL
LIN {X 0,Y 111.425,Z 449.114,A -85,B 0,C 180,E1 -28038.849,E2 -28038.849} C_VEL
LIN {X 0,Y 114.366,Z 436.579,A -85,B 0,C 180,E1 -28040.172,E2 -28040.172} C_VEL
LIN {X 0,Y 116.305,Z 423.133,A -85,B 0,C 180,E1 -28041.099,E2 -28041.099} C_VEL
LIN {X 0,Y 118.652,Z 397.035,A -85,B 0,C 180,E1 -28042.258,E2 -28042.258} C_VEL
LIN {X 0,Y 114.909,Z 388.618,A -85,B 0,C 180,E1 -28046.358,E2 -28046.358} C_VEL
LIN {X 0,Y 111.306,Z 381.772,A -85,B 0,C 180,E1 -28051.006,E2 -28051.006} C_VEL
LIN {X 0,Y 109.643,Z 378.864,A -85,B 0,C 180,E1 -28053.536,E2 -28053.536} C_VEL
LIN {X 0,Y 107.724,Z 375.644,A -85,B 0,C 180,E1 -28056.954,E2 -28056.954} C_VEL
LIN {X 0,Y 105.555,Z 371.862,A -85,B 0,C 180,E1 -28062.064,E2 -28062.064} C_VEL
LIN {X 0,Y 103.625,Z 368.788,A -85,B 0,C 180,E1 -28069.99,E2 -28069.99} C_VEL
LIN {X 0,Y 103.472,Z 367.177,A -85,B 0,C 180,E1 -28073.076,E2 -28073.076} C_VEL
LIN {X 0,Y 103.57,Z 367.162,A -85,B 0,C 180,E1 -28078.448,E2 -28078.448} C_VEL
LIN {X 0,Y 104.595,Z 370.555,A -85,B 0,C 180,E1 -28085.3,E2 -28085.3} C_VEL
LIN {X 0,Y 105.77,Z 371.985,A -85,B 0,C 180,E1 -28088.831,E2 -28088.831} C_VEL
LIN {X 0,Y 107.658,Z 375.474,A -85,B 0,C 180,E1 -28093.263,E2 -28093.263} C_VEL
LIN {X 0,Y 108.637,Z 377.169,A -85,B 0,C 180,E1 -28095.116,E2 -28095.116} C_VEL
LIN {X 0,Y 110.867,Z 380.964,A -85,B 0,C 180,E1 -28098.718,E2 -28098.718} C_VEL
LIN {X 0,Y 113.582,Z 385.928,A -85,B 0,C 180,E1 -28102.39,E2 -28102.39} C_VEL
LIN {X 0,Y 115.676,Z 390.593,A -85,B 0,C 180,E1 -28104.943,E2 -28104.943} C_VEL
LIN {X 0,Y 118.28,Z 399.597,A -85,B 0,C 180,E1 -28108.109,E2 -28108.109} C_VEL
LIN {X 0,Y 118.467,Z 401.333,A -85,B 0,C 180,E1 -28108.441,E2 -28108.441} C_VEL
LIN {X 0,Y 115.28,Z 434.09,A -85,B 0,C 180,E1 -28109.875,E2 -28109.875} C_VEL
LIN {X 0,Y 112.89,Z 447.226,A -85,B 0,C 180,E1 -28110.908,E2 -28110.908} C_VEL
LIN {X 0,Y 109.259,Z 460.289,A -85,B 0,C 180,E1 -28112.403,E2 -28112.403} C_VEL
LIN {X 0,Y 104.452,Z 472.907,A -85,B 0,C 180,E1 -28114.485,E2 -28114.485} C_VEL
LIN {X 0,Y 99.324,Z 484.193,A -85,B 0,C 180,E1 -28117.243,E2 -28117.243} C_VEL
LIN {X 0,Y 94.397,Z 493.302,A -85,B 0,C 180,E1 -28120.255,E2 -28120.255} C_VEL
LIN {X 0,Y 88.678,Z 502.639,A -85,B 0,C 180,E1 -28124.494,E2 -28124.494} C_VEL
LIN {X 0,Y 83.684,Z 510.076,A -85,B 0,C 180,E1 -28129.098,E2 -28129.098} C_VEL
LIN {X 0,Y 81.493,Z 513.266,A -85,B 0,C 180,E1 -28131.566,E2 -28131.566} C_VEL
LIN {X 0,Y 76.923,Z 520.058,A -85,B 0,C 180,E1 -28138.305,E2 -28138.305} C_VEL
LIN {X 0,Y 72.653,Z 526.459,A -85,B 0,C 180,E1 -28147.232,E2 -28147.232} C_VEL
LIN {X 0,Y 70.609,Z 530.652,A -85,B 0,C 180,E1 -28155.588,E2 -28155.588} C_VEL
LIN {X 0,Y 69.884,Z 533.758,A -85,B 0,C 180,E1 -28164.225,E2 -28164.225} C_VEL
LIN {X 0,Y 70.068,Z 535.289,A -85,B 0,C 180,E1 -28169.996,E2 -28169.996} C_VEL
LIN {X 0,Y 69.842,Z 536.305,A -85,B 0,C 180,E1 -28175.772,E2 -28175.772} C_VEL
LIN {X 0,Y 70.241,Z 536.926,A -85,B 0,C 180,E1 -28181.54,E2 -28181.54} C_VEL
LIN {X 0,Y 72.836,Z 537.025,A -85,B 0,C 180,E1 -28192.7,E2 -28192.7} C_VEL
LIN {X 0,Y 75.075,Z 536.474,A -85,B 0,C 180,E1 -28197.905,E2 -28197.905} C_VEL
LIN {X 0,Y 81.419,Z 534.194,A -85,B 0,C 180,E1 -28207.17,E2 -28207.17} C_VEL
LIN {X 0,Y 87.378,Z 531.412,A -85,B 0,C 180,E1 -28213.127,E2 -28213.127} C_VEL
LIN {X 0,Y 94.125,Z 527.632,A -85,B 0,C 180,E1 -28218.298,E2 -28218.298} C_VEL
LIN {X 0,Y 101.56,Z 522.759,A -85,B 0,C 180,E1 -28222.727,E2 -28222.727} C_VEL
LIN {X 0,Y 109.612,Z 516.646,A -85,B 0,C 180,E1 -28226.458,E2 -28226.458} C_VEL
LIN {X 0,Y 118.116,Z 509.073,A -85,B 0,C 180,E1 -28229.624,E2 -28229.624} C_VEL
LIN {X 0,Y 125.438,Z 501.358,A -85,B 0,C 180,E1 -28231.933,E2 -28231.933} C_VEL
LIN {X 0,Y 133.766,Z 490.904,A -85,B 0,C 180,E1 -28234.12,E2 -28234.12} C_VEL
LIN {X 0,Y 140.773,Z 480.276,A -85,B 0,C 180,E1 -28235.656,E2 -28235.656} C_VEL
LIN {X 0,Y 146.262,Z 470.027,A -85,B 0,C 180,E1 -28236.772,E2 -28236.772} C_VEL
LIN {X 0,Y 151.446,Z 457.842,A -85,B 0,C 180,E1 -28237.697,E2 -28237.697} C_VEL
LIN {X 0,Y 155.5,Z 444.729,A -85,B 0,C 180,E1 -28238.433,E2 -28238.433} C_VEL
LIN {X 0,Y 157.796,Z 433.749,A -85,B 0,C 180,E1 -28238.893,E2 -28238.893} C_VEL
LIN {X 0,Y 156.394,Z 427.276,A -85,B 0,C 180,E1 -28242.174,E2 -28242.174} C_VEL
LIN {X 0,Y 155.292,Z 423.303,A -85,B 0,C 180,E1 -28244.917,E2 -28244.917} C_VEL
LIN {X 0,Y 153.996,Z 420.252,A -85,B 0,C 180,E1 -28248.817,E2 -28248.817} C_VEL
LIN {X 0,Y 153.196,Z 417.427,A -85,B 0,C 180,E1 -28254.736,E2 -28254.736} C_VEL
LIN {X 0,Y 153.225,Z 417.62,A -85,B 0,C 180,E1 -28257.701,E2 -28257.701} C_VEL
LIN {X 0,Y 154.252,Z 420.509,A -85,B 0,C 180,E1 -28263.677,E2 -28263.677} C_VEL
LIN {X 0,Y 155.756,Z 424.425,A -85,B 0,C 180,E1 -28267.927,E2 -28267.927} C_VEL
LIN {X 0,Y 155.898,Z 424.798,A -85,B 0,C 180,E1 -28268.261,E2 -28268.261} C_VEL
LIN {X 0,Y 156.254,Z 427.053,A -85,B 0,C 180,E1 -28269.368,E2 -28269.368} C_VEL
LIN {X 0,Y 156.204,Z 430.198,A -85,B 0,C 180,E1 -28270.175,E2 -28270.175} C_VEL
LIN {X 0,Y 155.83,Z 433.855,A -85,B 0,C 180,E1 -28270.727,E2 -28270.727} C_VEL
LIN {X 0,Y 155.107,Z 437.675,A -85,B 0,C 180,E1 -28271.043,E2 -28271.043} C_VEL
LIN {X 0,Y 152.625,Z 446.309,A -85,B 0,C 180,E1 -28271.264,E2 -28271.264} C_VEL
LIN {X 0,Y 149.637,Z 454.644,A -85,B 0,C 180,E1 -28271.561,E2 -28271.561} C_VEL
LIN {X 0,Y 144.842,Z 465.728,A -85,B 0,C 180,E1 -28272.454,E2 -28272.454} C_VEL
LIN {X 0,Y 139.192,Z 476.12,A -85,B 0,C 180,E1 -28273.608,E2 -28273.608} C_VEL
LIN {X 0,Y 132.843,Z 485.761,A -85,B 0,C 180,E1 -28275.099,E2 -28275.099} C_VEL
LIN {X 0,Y 125.094,Z 495.574,A -85,B 0,C 180,E1 -28277.244,E2 -28277.244} C_VEL
LIN {X 0,Y 117.473,Z 503.569,A -85,B 0,C 180,E1 -28279.57,E2 -28279.57} C_VEL
LIN {X 0,Y 110.041,Z 510.164,A -85,B 0,C 180,E1 -28282.18,E2 -28282.18} C_VEL
LIN {X 0,Y 101.483,Z 516.606,A -85,B 0,C 180,E1 -28285.81,E2 -28285.81} C_VEL
LIN {X 0,Y 93.355,Z 521.678,A -85,B 0,C 180,E1 -28290.038,E2 -28290.038} C_VEL
LIN {X 0,Y 85.808,Z 525.582,A -85,B 0,C 180,E1 -28295.017,E2 -28295.017} C_VEL
LIN {X 0,Y 81.176,Z 527.573,A -85,B 0,C 180,E1 -28298.818,E2 -28298.818} C_VEL
LIN {X 0,Y 76.909,Z 529.14,A -85,B 0,C 180,E1 -28303.031,E2 -28303.031} C_VEL
LIN {X 0,Y 73.131,Z 530.282,A -85,B 0,C 180,E1 -28307.728,E2 -28307.728} C_VEL
LIN {X 0,Y 67.124,Z 531.271,A -85,B 0,C 180,E1 -28318.437,E2 -28318.437} C_VEL
LIN {X 0,Y 64.992,Z 531.183,A -85,B 0,C 180,E1 -28324.375,E2 -28324.375} C_VEL
LIN {X 0,Y 63.524,Z 530.687,A -85,B 0,C 180,E1 -28330.62,E2 -28330.62} C_VEL
LIN {X 0,Y 62.748,Z 528.433,A -85,B 0,C 180,E1 -28343.573,E2 -28343.573} C_VEL
LIN {X 0,Y 63.343,Z 526.714,A -85,B 0,C 180,E1 -28350.004,E2 -28350.004} C_VEL
LIN {X 0,Y 65.12,Z 523.298,A -85,B 0,C 180,E1 -28359.32,E2 -28359.32} C_VEL
LIN {X 0,Y 68.273,Z 518.815,A -85,B 0,C 180,E1 -28367.992,E2 -28367.992} C_VEL
LIN {X 0,Y 73.538,Z 512.024,A -85,B 0,C 180,E1 -28377.002,E2 -28377.002} C_VEL
LIN {X 0,Y 79.136,Z 504.662,A -85,B 0,C 180,E1 -28383.718,E2 -28383.718} C_VEL
LIN {X 0,Y 85.656,Z 495.497,A -85,B 0,C 180,E1 -28389.489,E2 -28389.489} C_VEL
LIN {X 0,Y 92.308,Z 484.895,A -85,B 0,C 180,E1 -28394.01,E2 -28394.01} C_VEL
LIN {X 0,Y 98.07,Z 474.09,A -85,B 0,C 180,E1 -28397.273,E2 -28397.273} C_VEL
LIN {X 0,Y 102.626,Z 463.563,A -85,B 0,C 180,E1 -28399.632,E2 -28399.632} C_VEL
LIN {X 0,Y 106.912,Z 450.937,A -85,B 0,C 180,E1 -28401.699,E2 -28401.699} C_VEL
LIN {X 0,Y 110.143,Z 438.317,A -85,B 0,C 180,E1 -28403.08,E2 -28403.08} C_VEL
LIN {X 0,Y 112.158,Z 426.211,A -85,B 0,C 180,E1 -28403.96,E2 -28403.96} C_VEL
LIN {X 0,Y 114.695,Z 399.913,A -85,B 0,C 180,E1 -28405.123,E2 -28405.123} C_VEL
LIN {X 0,Y 111.623,Z 392.88,A -85,B 0,C 180,E1 -28408.996,E2 -28408.996} C_VEL
LIN {X 0,Y 108.926,Z 387.374,A -85,B 0,C 180,E1 -28412.993,E2 -28412.993} C_VEL
LIN {X 0,Y 107.25,Z 384.249,A -85,B 0,C 180,E1 -28415.932,E2 -28415.932} C_VEL
LIN {X 0,Y 106.141,Z 382.164,A -85,B 0,C 180,E1 -28418.209,E2 -28418.209} C_VEL
LIN {X 0,Y 104.312,Z 378.721,A -85,B 0,C 180,E1 -28422.982,E2 -28422.982} C_VEL
LIN {X 0,Y 102.632,Z 375.543,A -85,B 0,C 180,E1 -28431.071,E2 -28431.071} C_VEL
LIN {X 0,Y 102.565,Z 374.178,A -85,B 0,C 180,E1 -28433.904,E2 -28433.904} C_VEL
LIN {X 0,Y 102.639,Z 374.166,A -85,B 0,C 180,E1 -28437.708,E2 -28437.708} C_VEL
LIN {X 0,Y 103.809,Z 377.887,A -85,B 0,C 180,E1 -28445.706,E2 -28445.706} C_VEL
LIN {X 0,Y 104.486,Z 378.821,A -85,B 0,C 180,E1 -28447.852,E2 -28447.852} C_VEL
LIN {X 0,Y 106.792,Z 383.332,A -85,B 0,C 180,E1 -28453.515,E2 -28453.515} C_VEL
LIN {X 0,Y 108.862,Z 387.185,A -85,B 0,C 180,E1 -28457.251,E2 -28457.251} C_VEL
LIN {X 0,Y 111.083,Z 391.599,A -85,B 0,C 180,E1 -28460.605,E2 -28460.605} C_VEL
LIN {X 0,Y 112.697,Z 395.452,A -85,B 0,C 180,E1 -28462.818,E2 -28462.818} C_VEL
LIN {X 0,Y 114.603,Z 402.714,A -85,B 0,C 180,E1 -28465.508,E2 -28465.508} C_VEL
LIN {X 0,Y 111.514,Z 433.384,A -85,B 0,C 180,E1 -28466.833,E2 -28466.833} C_VEL
LIN {X 0,Y 109.032,Z 446.614,A -85,B 0,C 180,E1 -28467.837,E2 -28467.837} C_VEL
LIN {X 0,Y 105.602,Z 458.671,A -85,B 0,C 180,E1 -28469.129,E2 -28469.129} C_VEL
LIN {X 0,Y 101.314,Z 470.038,A -85,B 0,C 180,E1 -28470.854,E2 -28470.854} C_VEL
LIN {X 0,Y 95.785,Z 481.764,A -85,B 0,C 180,E1 -28473.419,E2 -28473.419} C_VEL
LIN {X 0,Y 89.898,Z 492.318,A -85,B 0,C 180,E1 -28476.739,E2 -28476.739} C_VEL
LIN {X 0,Y 83.817,Z 501.816,A -85,B 0,C 180,E1 -28481.002,E2 -28481.002} C_VEL
LIN {X 0,Y 77.752,Z 510.182,A -85,B 0,C 180,E1 -28486.311,E2 -28486.311} C_VEL
LIN {X 0,Y 75.236,Z 513.602,A -85,B 0,C 180,E1 -28489.16,E2 -28489.16} C_VEL
LIN {X 0,Y 70.151,Z 520.444,A -85,B 0,C 180,E1 -28496.559,E2 -28496.559} C_VEL
LIN {X 0,Y 66.116,Z 525.884,A -85,B 0,C 180,E1 -28504.833,E2 -28504.833} C_VEL
LIN {X 0,Y 63.726,Z 530.134,A -85,B 0,C 180,E1 -28513.991,E2 -28513.991} C_VEL
LIN {X 0,Y 62.8,Z 533.292,A -85,B 0,C 180,E1 -28523.57,E2 -28523.57} C_VEL
LIN {X 0,Y 62.954,Z 534.854,A -85,B 0,C 180,E1 -28529.996,E2 -28529.996} C_VEL
LIN {X 0,Y 62.772,Z 535.914,A -85,B 0,C 180,E1 -28536.424,E2 -28536.424} C_VEL
LIN {X 0,Y 63.275,Z 536.559,A -85,B 0,C 180,E1 -28542.831,E2 -28542.831} C_VEL
LIN {X 0,Y 66.301,Z 536.704,A -85,B 0,C 180,E1 -28555.084,E2 -28555.084} C_VEL
LIN {X 0,Y 68.861,Z 536.201,A -85,B 0,C 180,E1 -28560.68,E2 -28560.68} C_VEL
LIN {X 0,Y 75.862,Z 533.971,A -85,B 0,C 180,E1 -28570.424,E2 -28570.424} C_VEL
LIN {X 0,Y 83.27,Z 530.782,A -85,B 0,C 180,E1 -28577.318,E2 -28577.318} C_VEL
LIN {X 0,Y 92.099,Z 526.06,A -85,B 0,C 180,E1 -28583.245,E2 -28583.245} C_VEL
LIN {X 0,Y 101.564,Z 519.838,A -85,B 0,C 180,E1 -28587.954,E2 -28587.954} C_VEL
LIN {X 0,Y 110.246,Z 513.098,A -85,B 0,C 180,E1 -28591.223,E2 -28591.223} C_VEL
LIN {X 0,Y 119.228,Z 504.763,A -85,B 0,C 180,E1 -28594.012,E2 -28594.012} C_VEL
LIN {X 0,Y 126.922,Z 496.209,A -85,B 0,C 180,E1 -28596.009,E2 -28596.009} C_VEL
LIN {X 0,Y 134.035,Z 486.846,A -85,B 0,C 180,E1 -28597.536,E2 -28597.536} C_VEL
LIN {X 0,Y 141.191,Z 475.262,A -85,B 0,C 180,E1 -28598.952,E2 -28598.952} C_VEL
LIN {X 0,Y 146.873,Z 463.813,A -85,B 0,C 180,E1 -28599.891,E2 -28599.891} C_VEL
LIN {X 0,Y 151.415,Z 451.72,A -85,B 0,C 180,E1 -28600.632,E2 -28600.632} C_VEL
LIN {X 0,Y 154.948,Z 438.484,A -85,B 0,C 180,E1 -28601.207,E2 -28601.207} C_VEL
LIN {X 0,Y 155.199,Z 437.051,A -85,B 0,C 180,E1 -28601.349,E2 -28601.349} C_VEL
LIN {X 0,Y 154.266,Z 431.352,A -85,B 0,C 180,E1 -28604.645,E2 -28604.645} C_VEL
LIN {X 0,Y 153.742,Z 429.532,A -85,B 0,C 180,E1 -28606.283,E2 -28606.283} C_VEL
LIN {X 0,Y 152.905,Z 427.113,A -85,B 0,C 180,E1 -28609.406,E2 -28609.406} C_VEL
LIN {X 0,Y 152.297,Z 424.659,A -85,B 0,C 180,E1 -28614.705,E2 -28614.705} C_VEL
LIN {X 0,Y 152.318,Z 424.793,A -85,B 0,C 180,E1 -28617.687,E2 -28617.687} C_VEL
LIN {X 0,Y 153.063,Z 427.259,A -85,B 0,C 180,E1 -28622.962,E2 -28622.962} C_VEL
LIN {X 0,Y 154.157,Z 430.897,A -85,B 0,C 180,E1 -28627.038,E2 -28627.038} C_VEL
LIN {X 0,Y 155.33,Z 434.908,A -85,B 0,C 180,E1 -28630.387,E2 -28630.387} C_VEL
LIN {X 0,Y 152.368,Z 446.51,A -85,B 0,C 180,E1 -28630.998,E2 -28630.998} C_VEL
LIN {X 0,Y 149.637,Z 454.644,A -85,B 0,C 180,E1 -28631.561,E2 -28631.561} C_VEL
LIN {X 0,Y 147.323,Z 460.071,A -85,B 0,C 180,E1 -28631.722,E2 -28631.722} C_VEL
LIN {X 0,Y 142.476,Z 468.696,A -85,B 0,C 180,E1 -28631.342,E2 -28631.342} C_VEL
LIN {X 0,Y 137.015,Z 476.919,A -85,B 0,C 180,E1 -28631.075,E2 -28631.075} C_VEL
LIN {X 0,Y 133.729,Z 481.706,A -85,B 0,C 180,E1 -28631.465,E2 -28631.465} C_VEL
LIN {X 0,Y 125.715,Z 492.375,A -85,B 0,C 180,E1 -28633.369,E2 -28633.369} C_VEL
LIN {X 0,Y 118.381,Z 500.393,A -85,B 0,C 180,E1 -28635.272,E2 -28635.272} C_VEL
LIN {X 0,Y 108.882,Z 508.978,A -85,B 0,C 180,E1 -28638.12,E2 -28638.12} C_VEL
LIN {X 0,Y 100.011,Z 515.619,A -85,B 0,C 180,E1 -28641.399,E2 -28641.399} C_VEL
LIN {X 0,Y 89.943,Z 521.779,A -85,B 0,C 180,E1 -28646.033,E2 -28646.033} C_VEL
LIN {X 0,Y 81.312,Z 525.97,A -85,B 0,C 180,E1 -28651.24,E2 -28651.24} C_VEL
LIN {X 0,Y 72.152,Z 529.356,A -85,B 0,C 180,E1 -28658.814,E2 -28658.814} C_VEL
LIN {X 0,Y 67.929,Z 530.538,A -85,B 0,C 180,E1 -28663.601,E2 -28663.601} C_VEL
LIN {X 0,Y 62.568,Z 531.49,A -85,B 0,C 180,E1 -28671.842,E2 -28671.842} C_VEL
LIN {X 0,Y 58.569,Z 531.532,A -85,B 0,C 180,E1 -28681.321,E2 -28681.321} C_VEL
LIN {X 0,Y 56.766,Z 531.081,A -85,B 0,C 180,E1 -28688.202,E2 -28688.202} C_VEL
LIN {X 0,Y 55.779,Z 530.187,A -85,B 0,C 180,E1 -28695.409,E2 -28695.409} C_VEL
LIN {X 0,Y 56.227,Z 527.282,A -85,B 0,C 180,E1 -28709.643,E2 -28709.643} C_VEL
LIN {X 0,Y 58.139,Z 523.833,A -85,B 0,C 180,E1 -28720.451,E2 -28720.451} C_VEL
LIN {X 0,Y 61.55,Z 519.414,A -85,B 0,C 180,E1 -28730.037,E2 -28730.037} C_VEL
LIN {X 0,Y 66.38,Z 513.801,A -85,B 0,C 180,E1 -28738.457,E2 -28738.457} C_VEL
LIN {X 0,Y 72.32,Z 506.783,A -85,B 0,C 180,E1 -28745.671,E2 -28745.671} C_VEL
LIN {X 0,Y 79.082,Z 498.026,A -85,B 0,C 180,E1 -28751.804,E2 -28751.804} C_VEL
LIN {X 0,Y 86.062,Z 488.048,A -85,B 0,C 180,E1 -28756.452,E2 -28756.452} C_VEL
LIN {X 0,Y 92.04,Z 477.861,A -85,B 0,C 180,E1 -28759.785,E2 -28759.785} C_VEL
LIN {X 0,Y 97.527,Z 466.577,A -85,B 0,C 180,E1 -28762.441,E2 -28762.441} C_VEL
LIN {X 0,Y 101.983,Z 454.921,A -85,B 0,C 180,E1 -28764.497,E2 -28764.497} C_VEL
LIN {X 0,Y 105.653,Z 442.432,A -85,B 0,C 180,E1 -28765.949,E2 -28765.949} C_VEL
LIN {X 0,Y 108.373,Z 428.501,A -85,B 0,C 180,E1 -28767.027,E2 -28767.027} C_VEL
LIN {X 0,Y 111.025,Z 403.057,A -85,B 0,C 180,E1 -28768.164,E2 -28768.164} C_VEL
LIN {X 0,Y 108.467,Z 396.793,A -85,B 0,C 180,E1 -28771.98,E2 -28771.98} C_VEL
LIN {X 0,Y 106.053,Z 391.56,A -85,B 0,C 180,E1 -28776.311,E2 -28776.311} C_VEL
LIN {X 0,Y 104.428,Z 388.396,A -85,B 0,C 180,E1 -28779.938,E2 -28779.938} C_VEL
LIN {X 0,Y 103.029,Z 385.437,A -85,B 0,C 180,E1 -28784.165,E2 -28784.165} C_VEL
LIN {X 0,Y 101.674,Z 382.245,A -85,B 0,C 180,E1 -28792.278,E2 -28792.278} C_VEL
LIN {X 0,Y 101.682,Z 381.207,A -85,B 0,C 180,E1 -28794.398,E2 -28794.398} C_VEL
LIN {X 0,Y 101.725,Z 381.34,A -85,B 0,C 180,E1 -28797.321,E2 -28797.321} C_VEL
LIN {X 0,Y 102.927,Z 385.04,A -85,B 0,C 180,E1 -28805.755,E2 -28805.755} C_VEL
LIN {X 0,Y 103.294,Z 385.874,A -85,B 0,C 180,E1 -28807.083,E2 -28807.083} C_VEL
LIN {X 0,Y 105.17,Z 389.786,A -85,B 0,C 180,E1 -28812.175,E2 -28812.175} C_VEL
LIN {X 0,Y 107.502,Z 394.534,A -85,B 0,C 180,E1 -28816.741,E2 -28816.741} C_VEL
LIN {X 0,Y 109.751,Z 399.862,A -85,B 0,C 180,E1 -28820.376,E2 -28820.376} C_VEL
LIN {X 0,Y 111,Z 405.097,A -85,B 0,C 180,E1 -28822.461,E2 -28822.461} C_VEL
LIN {X 0,Y 107.929,Z 433.586,A -85,B 0,C 180,E1 -28823.631,E2 -28823.631} C_VEL
LIN {X 0,Y 105.343,Z 446.643,A -85,B 0,C 180,E1 -28824.594,E2 -28824.594} C_VEL
LIN {X 0,Y 101.578,Z 459.229,A -85,B 0,C 180,E1 -28825.908,E2 -28825.908} C_VEL
LIN {X 0,Y 97.114,Z 470.352,A -85,B 0,C 180,E1 -28827.556,E2 -28827.556} C_VEL
LIN {X 0,Y 91.333,Z 481.958,A -85,B 0,C 180,E1 -28830.034,E2 -28830.034} C_VEL
LIN {X 0,Y 85.143,Z 492.424,A -85,B 0,C 180,E1 -28833.3,E2 -28833.3} C_VEL
LIN {X 0,Y 79.306,Z 500.974,A -85,B 0,C 180,E1 -28837.096,E2 -28837.096} C_VEL
LIN {X 0,Y 73.325,Z 508.82,A -85,B 0,C 180,E1 -28841.979,E2 -28841.979} C_VEL
LIN {X 0,Y 68.972,Z 514.151,A -85,B 0,C 180,E1 -28846.539,E2 -28846.539} C_VEL
LIN {X 0,Y 64.295,Z 519.807,A -85,B 0,C 180,E1 -28853.039,E2 -28853.039} C_VEL
LIN {X 0,Y 59.727,Z 525.309,A -85,B 0,C 180,E1 -28861.917,E2 -28861.917} C_VEL
LIN {X 0,Y 56.894,Z 529.616,A -85,B 0,C 180,E1 -28872.007,E2 -28872.007} C_VEL
LIN {X 0,Y 55.729,Z 532.827,A -85,B 0,C 180,E1 -28882.751,E2 -28882.751} C_VEL
LIN {X 0,Y 55.854,Z 534.415,A -85,B 0,C 180,E1 -28889.995,E2 -28889.995} C_VEL
LIN {X 0,Y 55.729,Z 535.522,A -85,B 0,C 180,E1 -28897.24,E2 -28897.24} C_VEL
LIN {X 0,Y 56.362,Z 536.192,A -85,B 0,C 180,E1 -28904.436,E2 -28904.436} C_VEL
LIN {X 0,Y 59.908,Z 536.384,A -85,B 0,C 180,E1 -28917.981,E2 -28917.981} C_VEL
LIN {X 0,Y 62.844,Z 535.917,A -85,B 0,C 180,E1 -28923.993,E2 -28923.993} C_VEL
LIN {X 0,Y 70.59,Z 533.748,A -85,B 0,C 180,E1 -28934.176,E2 -28934.176} C_VEL
LIN {X 0,Y 79.32,Z 530.3,A -85,B 0,C 180,E1 -28941.669,E2 -28941.669} C_VEL
LIN {X 0,Y 88.014,Z 525.958,A -85,B 0,C 180,E1 -28946.97,E2 -28946.97} C_VEL
LIN {X 0,Y 97.978,Z 519.819,A -85,B 0,C 180,E1 -28951.48,E2 -28951.48} C_VEL
LIN {X 0,Y 107.013,Z 513.149,A -85,B 0,C 180,E1 -28954.552,E2 -28954.552} C_VEL
LIN {X 0,Y 116.3,Z 504.896,A -85,B 0,C 180,E1 -28957.149,E2 -28957.149} C_VEL
LIN {X 0,Y 124.215,Z 496.467,A -85,B 0,C 180,E1 -28958.991,E2 -28958.991} C_VEL
LIN {X 0,Y 131.496,Z 487.241,A -85,B 0,C 180,E1 -28960.384,E2 -28960.384} C_VEL
LIN {X 0,Y 138.804,Z 475.815,A -85,B 0,C 180,E1 -28961.682,E2 -28961.682} C_VEL
LIN {X 0,Y 144.597,Z 464.59,A -85,B 0,C 180,E1 -28962.521,E2 -28962.521} C_VEL
LIN {X 0,Y 149.212,Z 452.998,A -85,B 0,C 180,E1 -28963.194,E2 -28963.194} C_VEL
LIN {X 0,Y 152.71,Z 440.866,A -85,B 0,C 180,E1 -28963.712,E2 -28963.712} C_VEL
LIN {X 0,Y 152.321,Z 436.764,A -85,B 0,C 180,E1 -28966.356,E2 -28966.356} C_VEL
LIN {X 0,Y 151.557,Z 433.925,A -85,B 0,C 180,E1 -28969.986,E2 -28969.986} C_VEL
LIN {X 0,Y 151.147,Z 431.824,A -85,B 0,C 180,E1 -28974.665,E2 -28974.665} C_VEL
LIN {X 0,Y 151.144,Z 431.936,A -85,B 0,C 180,E1 -28977.669,E2 -28977.669} C_VEL
LIN {X 0,Y 151.632,Z 434.148,A -85,B 0,C 180,E1 -28982.491,E2 -28982.491} C_VEL
LIN {X 0,Y 152.38,Z 437.832,A -85,B 0,C 180,E1 -28986.622,E2 -28986.622} C_VEL
LIN {X 0,Y 152.73,Z 439.375,A -85,B 0,C 180,E1 -28988.027,E2 -28988.027} C_VEL
LIN {X 0,Y 149.281,Z 450.959,A -85,B 0,C 180,E1 -28988.649,E2 -28988.649} C_VEL
LIN {X 0,Y 144.152,Z 463.491,A -85,B 0,C 180,E1 -28989.516,E2 -28989.516} C_VEL
LIN {X 0,Y 138.478,Z 474.209,A -85,B 0,C 180,E1 -28990.491,E2 -28990.491} C_VEL
LIN {X 0,Y 133.729,Z 481.706,A -85,B 0,C 180,E1 -28991.465,E2 -28991.465} C_VEL
LIN {X 0,Y 130.244,Z 486.419,A -85,B 0,C 180,E1 -28991.95,E2 -28991.95} C_VEL
LIN {X 0,Y 123.567,Z 493.801,A -85,B 0,C 180,E1 -28992.064,E2 -28992.064} C_VEL
LIN {X 0,Y 116.407,Z 500.64,A -85,B 0,C 180,E1 -28992.272,E2 -28992.272} C_VEL
LIN {X 0,Y 112.187,Z 504.426,A -85,B 0,C 180,E1 -28992.982,E2 -28992.982} C_VEL
LIN {X 0,Y 102.272,Z 512.398,A -85,B 0,C 180,E1 -28995.843,E2 -28995.843} C_VEL
LIN {X 0,Y 93.012,Z 518.505,A -85,B 0,C 180,E1 -28999.187,E2 -28999.187} C_VEL
LIN {X 0,Y 84.087,Z 523.309,A -85,B 0,C 180,E1 -29003.172,E2 -29003.172} C_VEL
LIN {X 0,Y 77.003,Z 526.436,A -85,B 0,C 180,E1 -29007.153,E2 -29007.153} C_VEL
LIN {X 0,Y 67.839,Z 529.575,A -85,B 0,C 180,E1 -29014.033,E2 -29014.033} C_VEL
LIN {X 0,Y 63.152,Z 530.784,A -85,B 0,C 180,E1 -29018.837,E2 -29018.837} C_VEL
LIN {X 0,Y 56.514,Z 531.853,A -85,B 0,C 180,E1 -29028.261,E2 -29028.261} C_VEL
LIN {X 0,Y 52.359,Z 531.88,A -85,B 0,C 180,E1 -29037.532,E2 -29037.532} C_VEL
LIN {X 0,Y 50.136,Z 531.459,A -85,B 0,C 180,E1 -29045.137,E2 -29045.137} C_VEL
LIN {X 0,Y 48.857,Z 530.613,A -85,B 0,C 180,E1 -29053.285,E2 -29053.285} C_VEL
LIN {X 0,Y 49.115,Z 527.669,A -85,B 0,C 180,E1 -29070.005,E2 -29070.005} C_VEL
LIN {X 0,Y 51.187,Z 524.364,A -85,B 0,C 180,E1 -29081.89,E2 -29081.89} C_VEL
LIN {X 0,Y 54.926,Z 520.007,A -85,B 0,C 180,E1 -29092.578,E2 -29092.578} C_VEL
LIN {X 0,Y 60.251,Z 514.457,A -85,B 0,C 180,E1 -29101.667,E2 -29101.667} C_VEL
LIN {X 0,Y 66.698,Z 507.54,A -85,B 0,C 180,E1 -29109.219,E2 -29109.219} C_VEL
LIN {X 0,Y 73.958,Z 498.88,A -85,B 0,C 180,E1 -29115.46,E2 -29115.46} C_VEL
LIN {X 0,Y 80.671,Z 489.983,A -85,B 0,C 180,E1 -29119.671,E2 -29119.671} C_VEL
LIN {X 0,Y 86.928,Z 480.224,A -85,B 0,C 180,E1 -29122.981,E2 -29122.981} C_VEL
LIN {X 0,Y 92.694,Z 469.482,A -85,B 0,C 180,E1 -29125.547,E2 -29125.547} C_VEL
LIN {X 0,Y 97.721,Z 457.491,A -85,B 0,C 180,E1 -29127.682,E2 -29127.682} C_VEL
LIN {X 0,Y 101.808,Z 444.905,A -85,B 0,C 180,E1 -29129.18,E2 -29129.18} C_VEL
LIN {X 0,Y 104.653,Z 432.109,A -85,B 0,C 180,E1 -29130.232,E2 -29130.232} C_VEL
LIN {X 0,Y 106.715,Z 415.897,A -85,B 0,C 180,E1 -29130.979,E2 -29130.979} C_VEL
LIN {X 0,Y 107.662,Z 406.247,A -85,B 0,C 180,E1 -29131.408,E2 -29131.408} C_VEL
LIN {X 0,Y 105.236,Z 400.044,A -85,B 0,C 180,E1 -29135.854,E2 -29135.854} C_VEL
LIN {X 0,Y 103.758,Z 396.658,A -85,B 0,C 180,E1 -29139.168,E2 -29139.168} C_VEL
LIN {X 0,Y 102.395,Z 393.64,A -85,B 0,C 180,E1 -29143.068,E2 -29143.068} C_VEL
LIN {X 0,Y 101.744,Z 392.102,A -85,B 0,C 180,E1 -29145.557,E2 -29145.557} C_VEL
LIN {X 0,Y 100.761,Z 388.981,A -85,B 0,C 180,E1 -29153.441,E2 -29153.441} C_VEL
LIN {X 0,Y 100.81,Z 388.212,A -85,B 0,C 180,E1 -29154.9,E2 -29154.9} C_VEL
LIN {X 0,Y 100.822,Z 388.555,A -85,B 0,C 180,E1 -29157.112,E2 -29157.112} C_VEL
LIN {X 0,Y 101.982,Z 392.379,A -85,B 0,C 180,E1 -29165.684,E2 -29165.684} C_VEL
LIN {X 0,Y 103.563,Z 396.193,A -85,B 0,C 180,E1 -29170.693,E2 -29170.693} C_VEL
LIN {X 0,Y 105.465,Z 400.485,A -85,B 0,C 180,E1 -29174.949,E2 -29174.949} C_VEL
LIN {X 0,Y 107.147,Z 404.921,A -85,B 0,C 180,E1 -29178.091,E2 -29178.091} C_VEL
LIN {X 0,Y 107.688,Z 407.461,A -85,B 0,C 180,E1 -29179.18,E2 -29179.18} C_VEL
LIN {X 0,Y 104.838,Z 432.955,A -85,B 0,C 180,E1 -29180.189,E2 -29180.189} C_VEL
LIN {X 0,Y 102.142,Z 446.137,A -85,B 0,C 180,E1 -29181.093,E2 -29181.093} C_VEL
LIN {X 0,Y 98.286,Z 458.666,A -85,B 0,C 180,E1 -29182.31,E2 -29182.31} C_VEL
LIN {X 0,Y 93.264,Z 470.644,A -85,B 0,C 180,E1 -29183.973,E2 -29183.973} C_VEL
LIN {X 0,Y 87.232,Z 482.137,A -85,B 0,C 180,E1 -29186.317,E2 -29186.317} C_VEL
LIN {X 0,Y 80.73,Z 492.51,A -85,B 0,C 180,E1 -29189.47,E2 -29189.47} C_VEL
LIN {X 0,Y 73.868,Z 501.812,A -85,B 0,C 180,E1 -29193.637,E2 -29193.637} C_VEL
LIN {X 0,Y 66.862,Z 510.117,A -85,B 0,C 180,E1 -29199.098,E2 -29199.098} C_VEL
LIN {X 0,Y 60.71,Z 517.003,A -85,B 0,C 180,E1 -29206,E2 -29206} C_VEL
LIN {X 0,Y 55.114,Z 523.032,A -85,B 0,C 180,E1 -29214.977,E2 -29214.977} C_VEL
LIN {X 0,Y 51.05,Z 527.781,A -85,B 0,C 180,E1 -29225.601,E2 -29225.601} C_VEL
LIN {X 0,Y 48.946,Z 531.4,A -85,B 0,C 180,E1 -29237.557,E2 -29237.557} C_VEL
LIN {X 0,Y 48.763,Z 533.977,A -85,B 0,C 180,E1 -29249.995,E2 -29249.995} C_VEL
LIN {X 0,Y 48.675,Z 535.118,A -85,B 0,C 180,E1 -29258.296,E2 -29258.296} C_VEL
LIN {X 0,Y 49.493,Z 535.824,A -85,B 0,C 180,E1 -29266.494,E2 -29266.494} C_VEL
LIN {X 0,Y 53.707,Z 536.063,A -85,B 0,C 180,E1 -29281.557,E2 -29281.557} C_VEL
LIN {X 0,Y 61.134,Z 534.788,A -85,B 0,C 180,E1 -29293.606,E2 -29293.606} C_VEL
LIN {X 0,Y 70.638,Z 531.878,A -85,B 0,C 180,E1 -29302.739,E2 -29302.739} C_VEL
LIN {X 0,Y 78.67,Z 528.595,A -85,B 0,C 180,E1 -29308.062,E2 -29308.062} C_VEL
LIN {X 0,Y 87.272,Z 524.271,A -85,B 0,C 180,E1 -29312.347,E2 -29312.347} C_VEL
LIN {X 0,Y 97.886,Z 517.776,A -85,B 0,C 180,E1 -29316.259,E2 -29316.259} C_VEL
LIN {X 0,Y 107.328,Z 510.685,A -85,B 0,C 180,E1 -29318.919,E2 -29318.919} C_VEL
LIN {X 0,Y 116.943,Z 501.871,A -85,B 0,C 180,E1 -29321.173,E2 -29321.173} C_VEL
LIN {X 0,Y 125.958,Z 491.876,A -85,B 0,C 180,E1 -29322.839,E2 -29322.839} C_VEL
LIN {X 0,Y 133.437,Z 481.677,A -85,B 0,C 180,E1 -29323.983,E2 -29323.983} C_VEL
LIN {X 0,Y 139.256,Z 471.975,A -85,B 0,C 180,E1 -29324.835,E2 -29324.835} C_VEL
LIN {X 0,Y 145.16,Z 459.679,A -85,B 0,C 180,E1 -29325.529,E2 -29325.529} C_VEL
LIN {X 0,Y 149.517,Z 447.582,A -85,B 0,C 180,E1 -29326.062,E2 -29326.062} C_VEL
LIN {X 0,Y 150.338,Z 444.592,A -85,B 0,C 180,E1 -29326.217,E2 -29326.217} C_VEL
LIN {X 0,Y 150.206,Z 442.641,A -85,B 0,C 180,E1 -29327.846,E2 -29327.846} C_VEL
LIN {X 0,Y 149.928,Z 440.841,A -85,B 0,C 180,E1 -29330.148,E2 -29330.148} C_VEL
LIN {X 0,Y 149.613,Z 438.885,A -85,B 0,C 180,E1 -29334.61,E2 -29334.61} C_VEL
LIN {X 0,Y 149.592,Z 438.954,A -85,B 0,C 180,E1 -29337.645,E2 -29337.645} C_VEL
LIN {X 0,Y 149.803,Z 440.813,A -85,B 0,C 180,E1 -29341.849,E2 -29341.849} C_VEL
LIN {X 0,Y 150.142,Z 443.768,A -85,B 0,C 180,E1 -29345.373,E2 -29345.373} C_VEL
LIN {X 0,Y 149.319,Z 446.762,A -85,B 0,C 180,E1 -29345.719,E2 -29345.719} C_VEL
LIN {X 0,Y 144.536,Z 459.609,A -85,B 0,C 180,E1 -29346.47,E2 -29346.47} C_VEL
LIN {X 0,Y 139.041,Z 470.72,A -85,B 0,C 180,E1 -29347.281,E2 -29347.281} C_VEL
LIN {X 0,Y 132.321,Z 481.502,A -85,B 0,C 180,E1 -29348.427,E2 -29348.427} C_VEL
LIN {X 0,Y 125.431,Z 490.643,A -85,B 0,C 180,E1 -29349.856,E2 -29349.856} C_VEL
LIN {X 0,Y 116.685,Z 500.197,A -85,B 0,C 180,E1 -29351.845,E2 -29351.845} C_VEL
LIN {X 0,Y 112.187,Z 504.426,A -85,B 0,C 180,E1 -29352.982,E2 -29352.982} C_VEL
LIN {X 0,Y 107.813,Z 508.087,A -85,B 0,C 180,E1 -29353.792,E2 -29353.792} C_VEL
LIN {X 0,Y 99.67,Z 513.646,A -85,B 0,C 180,E1 -29354.412,E2 -29354.412} C_VEL
LIN {X 0,Y 91.145,Z 518.515,A -85,B 0,C 180,E1 -29355.248,E2 -29355.248} C_VEL
LIN {X 0,Y 86.225,Z 521.095,A -85,B 0,C 180,E1 -29356.546,E2 -29356.546} C_VEL
LIN {X 0,Y 75.464,Z 526.027,A -85,B 0,C 180,E1 -29361.37,E2 -29361.37} C_VEL
LIN {X 0,Y 69.625,Z 528.144,A -85,B 0,C 180,E1 -29364.714,E2 -29364.714} C_VEL
LIN {X 0,Y 64.065,Z 529.793,A -85,B 0,C 180,E1 -29368.653,E2 -29368.653} C_VEL
LIN {X 0,Y 58.866,Z 531.03,A -85,B 0,C 180,E1 -29373.317,E2 -29373.317} C_VEL
LIN {X 0,Y 50.773,Z 532.208,A -85,B 0,C 180,E1 -29383.8,E2 -29383.8} C_VEL
LIN {X 0,Y 46.425,Z 532.229,A -85,B 0,C 180,E1 -29392.739,E2 -29392.739} C_VEL
LIN {X 0,Y 43.694,Z 531.834,A -85,B 0,C 180,E1 -29401.156,E2 -29401.156} C_VEL
LIN {X 0,Y 41.998,Z 531.037,A -85,B 0,C 180,E1 -29410.453,E2 -29410.453} C_VEL
LIN {X 0,Y 41.396,Z 529.795,A -85,B 0,C 180,E1 -29420.232,E2 -29420.232} C_VEL
LIN {X 0,Y 42.204,Z 527.71,A -85,B 0,C 180,E1 -29432.301,E2 -29432.301} C_VEL
LIN {X 0,Y 45.434,Z 523.597,A -85,B 0,C 180,E1 -29448.027,E2 -29448.027} C_VEL
LIN {X 0,Y 50.302,Z 518.911,A -85,B 0,C 180,E1 -29459.281,E2 -29459.281} C_VEL
LIN {X 0,Y 57.739,Z 511.873,A -85,B 0,C 180,E1 -29469.725,E2 -29469.725} C_VEL
LIN {X 0,Y 65.182,Z 504.253,A -85,B 0,C 180,E1 -29476.707,E2 -29476.707} C_VEL
LIN {X 0,Y 71.966,Z 496.443,A -85,B 0,C 180,E1 -29481.382,E2 -29481.382} C_VEL
LIN {X 0,Y 79.926,Z 485.826,A -85,B 0,C 180,E1 -29485.529,E2 -29485.529} C_VEL
LIN {X 0,Y 86.644,Z 475.004,A -85,B 0,C 180,E1 -29488.402,E2 -29488.402} C_VEL
LIN {X 0,Y 92.658,Z 462.7,A -85,B 0,C 180,E1 -29490.728,E2 -29490.728} C_VEL
LIN {X 0,Y 97.06,Z 451.067,A -85,B 0,C 180,E1 -29492.312,E2 -29492.312} C_VEL
LIN {X 0,Y 100.732,Z 437.883,A -85,B 0,C 180,E1 -29493.479,E2 -29493.479} C_VEL
LIN {X 0,Y 102.943,Z 425.302,A -85,B 0,C 180,E1 -29494.201,E2 -29494.201} C_VEL
LIN {X 0,Y 104.63,Z 409.726,A -85,B 0,C 180,E1 -29494.843,E2 -29494.843} C_VEL
LIN {X 0,Y 102.799,Z 404.414,A -85,B 0,C 180,E1 -29499.096,E2 -29499.096} C_VEL
LIN {X 0,Y 101.428,Z 401.116,A -85,B 0,C 180,E1 -29503.132,E2 -29503.132} C_VEL
LIN {X 0,Y 100.722,Z 399.072,A -85,B 0,C 180,E1 -29506.075,E2 -29506.075} C_VEL
LIN {X 0,Y 99.883,Z 395.784,A -85,B 0,C 180,E1 -29514.486,E2 -29514.486} C_VEL
LIN {X 0,Y 99.942,Z 395.314,A -85,B 0,C 180,E1 -29515.967,E2 -29515.967} C_VEL
LIN {X 0,Y 100.801,Z 399.188,A -85,B 0,C 180,E1 -29524.623,E2 -29524.623} C_VEL
LIN {X 0,Y 102.194,Z 403.004,A -85,B 0,C 180,E1 -29529.649,E2 -29529.649} C_VEL
LIN {X 0,Y 103.76,Z 406.988,A -85,B 0,C 180,E1 -29533.588,E2 -29533.588} C_VEL
LIN {X 0,Y 104.724,Z 409.997,A -85,B 0,C 180,E1 -29535.709,E2 -29535.709} C_VEL
LIN {X 0,Y 102.005,Z 433.099,A -85,B 0,C 180,E1 -29536.588,E2 -29536.588} C_VEL
LIN {X 0,Y 99.133,Z 446.432,A -85,B 0,C 180,E1 -29537.443,E2 -29537.443} C_VEL
LIN {X 0,Y 95.005,Z 459.12,A -85,B 0,C 180,E1 -29538.585,E2 -29538.585} C_VEL
LIN {X 0,Y 89.813,Z 470.922,A -85,B 0,C 180,E1 -29540.104,E2 -29540.104} C_VEL
LIN {X 0,Y 83.533,Z 482.301,A -85,B 0,C 180,E1 -29542.251,E2 -29542.251} C_VEL
LIN {X 0,Y 76.718,Z 492.566,A -85,B 0,C 180,E1 -29545.219,E2 -29545.219} C_VEL
LIN {X 0,Y 68.752,Z 502.62,A -85,B 0,C 180,E1 -29549.663,E2 -29549.663} C_VEL
LIN {X 0,Y 61.886,Z 510.1,A -85,B 0,C 180,E1 -29554.596,E2 -29554.596} C_VEL
LIN {X 0,Y 54.62,Z 517.452,A -85,B 0,C 180,E1 -29562.274,E2 -29562.274} C_VEL
LIN {X 0,Y 49.435,Z 522.418,A -85,B 0,C 180,E1 -29570.22,E2 -29570.22} C_VEL
LIN {X 0,Y 44.644,Z 527.228,A -85,B 0,C 180,E1 -29581.812,E2 -29581.812} C_VEL
LIN {X 0,Y 42.014,Z 530.904,A -85,B 0,C 180,E1 -29595.462,E2 -29595.462} C_VEL
LIN {X 0,Y 41.643,Z 533.533,A -85,B 0,C 180,E1 -29609.994,E2 -29609.994} C_VEL
LIN {X 0,Y 41.647,Z 534.701,A -85,B 0,C 180,E1 -29619.709,E2 -29619.709} C_VEL
LIN {X 0,Y 42.717,Z 535.455,A -85,B 0,C 180,E1 -29629.205,E2 -29629.205} C_VEL
LIN {X 0,Y 47.772,Z 535.744,A -85,B 0,C 180,E1 -29646.041,E2 -29646.041} C_VEL
LIN {X 0,Y 56.18,Z 534.536,A -85,B 0,C 180,E1 -29658.634,E2 -29658.634} C_VEL
LIN {X 0,Y 66.555,Z 531.684,A -85,B 0,C 180,E1 -29667.641,E2 -29667.641} C_VEL
LIN {X 0,Y 75.147,Z 528.456,A -85,B 0,C 180,E1 -29672.675,E2 -29672.675} C_VEL
LIN {X 0,Y 84.209,Z 524.19,A -85,B 0,C 180,E1 -29676.635,E2 -29676.635} C_VEL
LIN {X 0,Y 95.245,Z 517.757,A -85,B 0,C 180,E1 -29680.179,E2 -29680.179} C_VEL
LIN {X 0,Y 104.984,Z 510.769,A -85,B 0,C 180,E1 -29682.534,E2 -29682.534} C_VEL
LIN {X 0,Y 114.853,Z 502.044,A -85,B 0,C 180,E1 -29684.52,E2 -29684.52} C_VEL
LIN {X 0,Y 123.213,Z 493.13,A -85,B 0,C 180,E1 -29685.844,E2 -29685.844} C_VEL
LIN {X 0,Y 130.825,Z 483.344,A -85,B 0,C 180,E1 -29686.818,E2 -29686.818} C_VEL
LIN {X 0,Y 137.573,Z 472.622,A -85,B 0,C 180,E1 -29687.682,E2 -29687.682} C_VEL
LIN {X 0,Y 143.557,Z 460.579,A -85,B 0,C 180,E1 -29688.263,E2 -29688.263} C_VEL
LIN {X 0,Y 147.617,Z 449.93,A -85,B 0,C 180,E1 -29688.697,E2 -29688.697} C_VEL
LIN {X 0,Y 147.901,Z 448.746,A -85,B 0,C 180,E1 -29689.044,E2 -29689.044} C_VEL
LIN {X 0,Y 147.708,Z 447.089,A -85,B 0,C 180,E1 -29691.794,E2 -29691.794} C_VEL
LIN {X 0,Y 147.683,Z 445.898,A -85,B 0,C 180,E1 -29694.539,E2 -29694.539} C_VEL
LIN {X 0,Y 147.685,Z 445.712,A -85,B 0,C 180,E1 -29697.273,E2 -29697.273} C_VEL
LIN {X 0,Y 147.632,Z 447.594,A -85,B 0,C 180,E1 -29701.467,E2 -29701.467} C_VEL
LIN {X 0,Y 147.64,Z 448.834,A -85,B 0,C 180,E1 -29703.07,E2 -29703.07} C_VEL
LIN {X 0,Y 143.528,Z 459.522,A -85,B 0,C 180,E1 -29703.666,E2 -29703.666} C_VEL
LIN {X 0,Y 137.452,Z 471.578,A -85,B 0,C 180,E1 -29704.431,E2 -29704.431} C_VEL
LIN {X 0,Y 130.603,Z 482.259,A -85,B 0,C 180,E1 -29705.447,E2 -29705.447} C_VEL
LIN {X 0,Y 122.423,Z 492.65,A -85,B 0,C 180,E1 -29706.944,E2 -29706.944} C_VEL
LIN {X 0,Y 113.745,Z 501.62,A -85,B 0,C 180,E1 -29708.676,E2 -29708.676} C_VEL
LIN {X 0,Y 103.806,Z 509.962,A -85,B 0,C 180,E1 -29710.992,E2 -29710.992} C_VEL
LIN {X 0,Y 94.073,Z 516.645,A -85,B 0,C 180,E1 -29713.795,E2 -29713.795} C_VEL
LIN {X 0,Y 86.225,Z 521.095,A -85,B 0,C 180,E1 -29716.546,E2 -29716.546} C_VEL
LIN {X 0,Y 81.246,Z 523.46,A -85,B 0,C 180,E1 -29718.036,E2 -29718.036} C_VEL
LIN {X 0,Y 72.198,Z 526.85,A -85,B 0,C 180,E1 -29719.744,E2 -29719.744} C_VEL
LIN {X 0,Y 63.036,Z 529.527,A -85,B 0,C 180,E1 -29722.037,E2 -29722.037} C_VEL
LIN {X 0,Y 58.013,Z 530.647,A -85,B 0,C 180,E1 -29724.749,E2 -29724.749} C_VEL
LIN {X 0,Y 49.897,Z 532.136,A -85,B 0,C 180,E1 -29732.326,E2 -29732.326} C_VEL
LIN {X 0,Y 45.079,Z 532.565,A -85,B 0,C 180,E1 -29738.793,E2 -29738.793} C_VEL
LIN {X 0,Y 37.539,Z 532.208,A -85,B 0,C 180,E1 -29755.838,E2 -29755.838} C_VEL
LIN {X 0,Y 35.29,Z 531.448,A -85,B 0,C 180,E1 -29766.536,E2 -29766.536} C_VEL
LIN {X 0,Y 34.333,Z 530.247,A -85,B 0,C 180,E1 -29778.195,E2 -29778.195} C_VEL
LIN {X 0,Y 35.238,Z 527.951,A -85,B 0,C 180,E1 -29794.23,E2 -29794.23} C_VEL
LIN {X 0,Y 38.761,Z 524.155,A -85,B 0,C 180,E1 -29811.269,E2 -29811.269} C_VEL
LIN {X 0,Y 44.237,Z 519.532,A -85,B 0,C 180,E1 -29823.79,E2 -29823.79} C_VEL
LIN {X 0,Y 52.486,Z 512.56,A -85,B 0,C 180,E1 -29834.674,E2 -29834.674} C_VEL
LIN {X 0,Y 60.556,Z 505.028,A -85,B 0,C 180,E1 -29841.578,E2 -29841.578} C_VEL
LIN {X 0,Y 67.777,Z 497.326,A -85,B 0,C 180,E1 -29846.058,E2 -29846.058} C_VEL
LIN {X 0,Y 76.152,Z 486.838,A -85,B 0,C 180,E1 -29849.913,E2 -29849.913} C_VEL
LIN {X 0,Y 83.156,Z 476.172,A -85,B 0,C 180,E1 -29852.556,E2 -29852.556} C_VEL
LIN {X 0,Y 88.631,Z 465.874,A -85,B 0,C 180,E1 -29854.427,E2 -29854.427} C_VEL
LIN {X 0,Y 93.53,Z 454.125,A -85,B 0,C 180,E1 -29856,E2 -29856} C_VEL
LIN {X 0,Y 97.644,Z 440.887,A -85,B 0,C 180,E1 -29857.129,E2 -29857.129} C_VEL
LIN {X 0,Y 100.303,Z 427.838,A -85,B 0,C 180,E1 -29857.876,E2 -29857.876} C_VEL
LIN {X 0,Y 101.985,Z 413.338,A -85,B 0,C 180,E1 -29858.458,E2 -29858.458} C_VEL
LIN {X 0,Y 100.769,Z 409.508,A -85,B 0,C 180,E1 -29862.102,E2 -29862.102} C_VEL
LIN {X 0,Y 99.572,Z 405.831,A -85,B 0,C 180,E1 -29867.256,E2 -29867.256} C_VEL
LIN {X 0,Y 99.039,Z 402.628,A -85,B 0,C 180,E1 -29875.93,E2 -29875.93} C_VEL
LIN {X 0,Y 99.68,Z 406.027,A -85,B 0,C 180,E1 -29883.647,E2 -29883.647} C_VEL
LIN {X 0,Y 100.769,Z 409.529,A -85,B 0,C 180,E1 -29888.27,E2 -29888.27} C_VEL
LIN {X 0,Y 102.086,Z 413.529,A -85,B 0,C 180,E1 -29892.137,E2 -29892.137} C_VEL
LIN {X 0,Y 99.565,Z 433.434,A -85,B 0,C 180,E1 -29892.809,E2 -29892.809} C_VEL
LIN {X 0,Y 96.676,Z 446.234,A -85,B 0,C 180,E1 -29893.539,E2 -29893.539} C_VEL
LIN {X 0,Y 92.568,Z 458.552,A -85,B 0,C 180,E1 -29894.521,E2 -29894.521} C_VEL
LIN {X 0,Y 86.799,Z 471.197,A -85,B 0,C 180,E1 -29895.939,E2 -29895.939} C_VEL
LIN {X 0,Y 80.293,Z 482.465,A -85,B 0,C 180,E1 -29897.835,E2 -29897.835} C_VEL
LIN {X 0,Y 73.174,Z 492.611,A -85,B 0,C 180,E1 -29900.528,E2 -29900.528} C_VEL
LIN {X 0,Y 65.499,Z 501.777,A -85,B 0,C 180,E1 -29904.202,E2 -29904.202} C_VEL
LIN {X 0,Y 57.351,Z 510.088,A -85,B 0,C 180,E1 -29909.35,E2 -29909.35} C_VEL
LIN {X 0,Y 50.096,Z 516.772,A -85,B 0,C 180,E1 -29916.219,E2 -29916.219} C_VEL
LIN {X 0,Y 44.187,Z 521.804,A -85,B 0,C 180,E1 -29924.288,E2 -29924.288} C_VEL
LIN {X 0,Y 38.487,Z 526.673,A -85,B 0,C 180,E1 -29936.774,E2 -29936.774} C_VEL
LIN {X 0,Y 35.168,Z 530.407,A -85,B 0,C 180,E1 -29952.549,E2 -29952.549} C_VEL
LIN {X 0,Y 34.55,Z 533.091,A -85,B 0,C 180,E1 -29969.993,E2 -29969.993} C_VEL
LIN {X 0,Y 34.669,Z 534.283,A -85,B 0,C 180,E1 -29981.688,E2 -29981.688} C_VEL
LIN {X 0,Y 36.052,Z 535.077,A -85,B 0,C 180,E1 -29992.939,E2 -29992.939} C_VEL
LIN {X 0,Y 42.213,Z 535.424,A -85,B 0,C 180,E1 -30011.748,E2 -30011.748} C_VEL
LIN {X 0,Y 51.741,Z 534.271,A -85,B 0,C 180,E1 -30024.576,E2 -30024.576} C_VEL
LIN {X 0,Y 57.239,Z 533.092,A -85,B 0,C 180,E1 -30029.25,E2 -30029.25} C_VEL
LIN {X 0,Y 69.054,Z 529.485,A -85,B 0,C 180,E1 -30036.335,E2 -30036.335} C_VEL
LIN {X 0,Y 78.445,Z 525.628,A -85,B 0,C 180,E1 -30040.162,E2 -30040.162} C_VEL
LIN {X 0,Y 88.144,Z 520.673,A -85,B 0,C 180,E1 -30043.087,E2 -30043.087} C_VEL
LIN {X 0,Y 98.064,Z 514.468,A -85,B 0,C 180,E1 -30045.344,E2 -30045.344} C_VEL
LIN {X 0,Y 108.102,Z 506.772,A -85,B 0,C 180,E1 -30047.2,E2 -30047.2} C_VEL
LIN {X 0,Y 116.582,Z 498.915,A -85,B 0,C 180,E1 -30048.4,E2 -30048.4} C_VEL
LIN {X 0,Y 125.11,Z 489.345,A -85,B 0,C 180,E1 -30049.425,E2 -30049.425} C_VEL
LIN {X 0,Y 132.807,Z 478.752,A -85,B 0,C 180,E1 -30050.257,E2 -30050.257} C_VEL
LIN {X 0,Y 138.543,Z 469.066,A -85,B 0,C 180,E1 -30050.757,E2 -30050.757} C_VEL
LIN {X 0,Y 143.831,Z 457.922,A -85,B 0,C 180,E1 -30051.187,E2 -30051.187} C_VEL
LIN {X 0,Y 144.623,Z 455.941,A -85,B 0,C 180,E1 -30051.257,E2 -30051.257} C_VEL
LIN {X 0,Y 145.29,Z 453.997,A -85,B 0,C 180,E1 -30051.657,E2 -30051.657} C_VEL
LIN {X 0,Y 145.339,Z 452.732,A -85,B 0,C 180,E1 -30054.451,E2 -30054.451} C_VEL
LIN {X 0,Y 145.343,Z 452.487,A -85,B 0,C 180,E1 -30057.229,E2 -30057.229} C_VEL
LIN {X 0,Y 145.16,Z 453.787,A -85,B 0,C 180,E1 -30060.367,E2 -30060.367} C_VEL
LIN {X 0,Y 144.846,Z 454.714,A -85,B 0,C 180,E1 -30060.635,E2 -30060.635} C_VEL
LIN {X 0,Y 139.706,Z 466.115,A -85,B 0,C 180,E1 -30061.174,E2 -30061.174} C_VEL
LIN {X 0,Y 133.595,Z 476.697,A -85,B 0,C 180,E1 -30061.824,E2 -30061.824} C_VEL
LIN {X 0,Y 125.536,Z 487.858,A -85,B 0,C 180,E1 -30062.925,E2 -30062.925} C_VEL
LIN {X 0,Y 118.028,Z 496.389,A -85,B 0,C 180,E1 -30064.18,E2 -30064.18} C_VEL
LIN {X 0,Y 109.465,Z 504.469,A -85,B 0,C 180,E1 -30065.669,E2 -30065.669} C_VEL
LIN {X 0,Y 99.298,Z 512.341,A -85,B 0,C 180,E1 -30067.766,E2 -30067.766} C_VEL
LIN {X 0,Y 89.299,Z 518.586,A -85,B 0,C 180,E1 -30070.351,E2 -30070.351} C_VEL
LIN {X 0,Y 79.507,Z 523.517,A -85,B 0,C 180,E1 -30073.52,E2 -30073.52} C_VEL
LIN {X 0,Y 69.961,Z 527.306,A -85,B 0,C 180,E1 -30077.541,E2 -30077.541} C_VEL
LIN {X 0,Y 60.926,Z 530.011,A -85,B 0,C 180,E1 -30082.667,E2 -30082.667} C_VEL
LIN {X 0,Y 58.013,Z 530.647,A -85,B 0,C 180,E1 -30084.749,E2 -30084.749} C_VEL
LIN {X 0,Y 53.096,Z 531.645,A -85,B 0,C 180,E1 -30087.992,E2 -30087.992} C_VEL
LIN {X 0,Y 44.227,Z 532.635,A -85,B 0,C 180,E1 -30093.1,E2 -30093.1} C_VEL
LIN {X 0,Y 37.342,Z 532.906,A -85,B 0,C 180,E1 -30098.722,E2 -30098.722} C_VEL
LIN {X 0,Y 33.04,Z 532.738,A -85,B 0,C 180,E1 -30105.37,E2 -30105.37} C_VEL
LIN {X 0,Y 31.927,Z 532.592,A -85,B 0,C 180,E1 -30108.247,E2 -30108.247} C_VEL
LIN {X 0,Y 28.835,Z 531.848,A -85,B 0,C 180,E1 -30120.836,E2 -30120.836} C_VEL
LIN {X 0,Y 27.33,Z 530.7,A -85,B 0,C 180,E1 -30135.108,E2 -30135.108} C_VEL
LIN {X 0,Y 28.339,Z 528.168,A -85,B 0,C 180,E1 -30157.23,E2 -30157.23} C_VEL
LIN {X 0,Y 32.261,Z 524.703,A -85,B 0,C 180,E1 -30175.838,E2 -30175.838} C_VEL
LIN {X 0,Y 38.532,Z 520.148,A -85,B 0,C 180,E1 -30189.68,E2 -30189.68} C_VEL
LIN {X 0,Y 47.712,Z 513.247,A -85,B 0,C 180,E1 -30200.662,E2 -30200.662} C_VEL
LIN {X 0,Y 56.439,Z 505.789,A -85,B 0,C 180,E1 -30207.205,E2 -30207.205} C_VEL
LIN {X 0,Y 64.099,Z 498.179,A -85,B 0,C 180,E1 -30211.309,E2 -30211.309} C_VEL
LIN {X 0,Y 72.047,Z 488.922,A -85,B 0,C 180,E1 -30214.472,E2 -30214.472} C_VEL
LIN {X 0,Y 79.326,Z 478.617,A -85,B 0,C 180,E1 -30216.815,E2 -30216.815} C_VEL
LIN {X 0,Y 85.828,Z 467.212,A -85,B 0,C 180,E1 -30218.669,E2 -30218.669} C_VEL
LIN {X 0,Y 90.914,Z 455.801,A -85,B 0,C 180,E1 -30220.069,E2 -30220.069} C_VEL
LIN {X 0,Y 95.14,Z 443.124,A -85,B 0,C 180,E1 -30221.036,E2 -30221.036} C_VEL
LIN {X 0,Y 98.037,Z 430.285,A -85,B 0,C 180,E1 -30221.707,E2 -30221.707} C_VEL
LIN {X 0,Y 99.732,Z 417.254,A -85,B 0,C 180,E1 -30222.24,E2 -30222.24} C_VEL
LIN {X 0,Y 98.887,Z 414.234,A -85,B 0,C 180,E1 -30225.858,E2 -30225.858} C_VEL
LIN {X 0,Y 98.437,Z 412.487,A -85,B 0,C 180,E1 -30228.676,E2 -30228.676} C_VEL
LIN {X 0,Y 98.141,Z 409.904,A -85,B 0,C 180,E1 -30235.892,E2 -30235.892} C_VEL
LIN {X 0,Y 98.556,Z 412.734,A -85,B 0,C 180,E1 -30242.426,E2 -30242.426} C_VEL
LIN {X 0,Y 99.371,Z 415.967,A -85,B 0,C 180,E1 -30246.726,E2 -30246.726} C_VEL
LIN {X 0,Y 99.804,Z 417.441,A -85,B 0,C 180,E1 -30248.363,E2 -30248.363} C_VEL
LIN {X 0,Y 97.559,Z 433.871,A -85,B 0,C 180,E1 -30248.858,E2 -30248.858} C_VEL
LIN {X 0,Y 94.634,Z 446.249,A -85,B 0,C 180,E1 -30249.468,E2 -30249.468} C_VEL
LIN {X 0,Y 90.622,Z 457.979,A -85,B 0,C 180,E1 -30250.263,E2 -30250.263} C_VEL
LIN {X 0,Y 85.122,Z 469.884,A -85,B 0,C 180,E1 -30251.334,E2 -30251.334} C_VEL
LIN {X 0,Y 78.405,Z 481.33,A -85,B 0,C 180,E1 -30252.876,E2 -30252.876} C_VEL
LIN {X 0,Y 70.987,Z 491.666,A -85,B 0,C 180,E1 -30255.127,E2 -30255.127} C_VEL
LIN {X 0,Y 62.909,Z 500.937,A -85,B 0,C 180,E1 -30258.257,E2 -30258.257} C_VEL
LIN {X 0,Y 55.088,Z 508.588,A -85,B 0,C 180,E1 -30262.33,E2 -30262.33} C_VEL
LIN {X 0,Y 49.563,Z 513.342,A -85,B 0,C 180,E1 -30266.007,E2 -30266.007} C_VEL
LIN {X 0,Y 42.136,Z 519.273,A -85,B 0,C 180,E1 -30273.48,E2 -30273.48} C_VEL
LIN {X 0,Y 34.774,Z 524.62,A -85,B 0,C 180,E1 -30284.969,E2 -30284.969} C_VEL
LIN {X 0,Y 29.524,Z 528.779,A -85,B 0,C 180,E1 -30301.56,E2 -30301.56} C_VEL
LIN {X 0,Y 27.696,Z 530.953,A -85,B 0,C 180,E1 -30315.291,E2 -30315.291} C_VEL
LIN {X 0,Y 27.45,Z 532.648,A -85,B 0,C 180,E1 -30329.991,E2 -30329.991} C_VEL
LIN {X 0,Y 27.74,Z 533.865,A -85,B 0,C 180,E1 -30344.666,E2 -30344.666} C_VEL
LIN {X 0,Y 29.618,Z 534.688,A -85,B 0,C 180,E1 -30358.322,E2 -30358.322} C_VEL
LIN {X 0,Y 32.874,Z 535.098,A -85,B 0,C 180,E1 -30369.884,E2 -30369.884} C_VEL
LIN {X 0,Y 42.333,Z 534.741,A -85,B 0,C 180,E1 -30386.096,E2 -30386.096} C_VEL
LIN {X 0,Y 53.948,Z 532.871,A -85,B 0,C 180,E1 -30395.76,E2 -30395.76} C_VEL
LIN {X 0,Y 66.513,Z 529.318,A -85,B 0,C 180,E1 -30401.973,E2 -30401.973} C_VEL
LIN {X 0,Y 76.327,Z 525.518,A -85,B 0,C 180,E1 -30405.184,E2 -30405.184} C_VEL
LIN {X 0,Y 86.342,Z 520.622,A -85,B 0,C 180,E1 -30407.612,E2 -30407.612} C_VEL
LIN {X 0,Y 96.512,Z 514.484,A -85,B 0,C 180,E1 -30409.429,E2 -30409.429} C_VEL
LIN {X 0,Y 106.757,Z 506.881,A -85,B 0,C 180,E1 -30410.908,E2 -30410.908} C_VEL
LIN {X 0,Y 115.366,Z 499.125,A -85,B 0,C 180,E1 -30411.847,E2 -30411.847} C_VEL
LIN {X 0,Y 124.006,Z 489.677,A -85,B 0,C 180,E1 -30412.643,E2 -30412.643} C_VEL
LIN {X 0,Y 131.795,Z 479.221,A -85,B 0,C 180,E1 -30413.291,E2 -30413.291} C_VEL
LIN {X 0,Y 138.107,Z 468.765,A -85,B 0,C 180,E1 -30413.698,E2 -30413.698} C_VEL
LIN {X 0,Y 142.028,Z 460.856,A -85,B 0,C 180,E1 -30413.925,E2 -30413.925} C_VEL
LIN {X 0,Y 142.601,Z 459.452,A -85,B 0,C 180,E1 -30414.344,E2 -30414.344} C_VEL
LIN {X 0,Y 142.626,Z 459.122,A -85,B 0,C 180,E1 -30417.176,E2 -30417.176} C_VEL
LIN {X 0,Y 142.547,Z 459.356,A -85,B 0,C 180,E1 -30417.812,E2 -30417.812} C_VEL
LIN {X 0,Y 142.056,Z 460.496,A -85,B 0,C 180,E1 -30418.023,E2 -30418.023} C_VEL
LIN {X 0,Y 136.111,Z 471.992,A -85,B 0,C 180,E1 -30418.51,E2 -30418.51} C_VEL
LIN {X 0,Y 129.147,Z 482.586,A -85,B 0,C 180,E1 -30419.208,E2 -30419.208} C_VEL
LIN {X 0,Y 121.277,Z 492.323,A -85,B 0,C 180,E1 -30420.172,E2 -30420.172} C_VEL
LIN {X 0,Y 112.476,Z 501.253,A -85,B 0,C 180,E1 -30421.384,E2 -30421.384} C_VEL
LIN {X 0,Y 103.774,Z 508.536,A -85,B 0,C 180,E1 -30422.701,E2 -30422.701} C_VEL
LIN {X 0,Y 94.084,Z 515.241,A -85,B 0,C 180,E1 -30424.461,E2 -30424.461} C_VEL
LIN {X 0,Y 84.881,Z 520.442,A -85,B 0,C 180,E1 -30426.522,E2 -30426.522} C_VEL
LIN {X 0,Y 74.788,Z 525.042,A -85,B 0,C 180,E1 -30429.374,E2 -30429.374} C_VEL
LIN {X 0,Y 64.918,Z 528.51,A -85,B 0,C 180,E1 -30433.025,E2 -30433.025} C_VEL
LIN {X 0,Y 54.071,Z 531.151,A -85,B 0,C 180,E1 -30438.745,E2 -30438.745} C_VEL
LIN {X 0,Y 46.427,Z 532.408,A -85,B 0,C 180,E1 -30444.745,E2 -30444.745} C_VEL
LIN {X 0,Y 40.607,Z 532.896,A -85,B 0,C 180,E1 -30451.284,E2 -30451.284} C_VEL
LIN {X 0,Y 31.927,Z 532.592,A -85,B 0,C 180,E1 -30468.247,E2 -30468.247} C_VEL
LIN {X 0,Y 28.75,Z 532.133,A -85,B 0,C 180,E1 -30477.622,E2 -30477.622} C_VEL
LIN {X 0,Y 23.791,Z 530.691,A -85,B 0,C 180,E1 -30496.231,E2 -30496.231} C_VEL
LIN {X 0,Y 21.912,Z 528.979,A -85,B 0,C 180,E1 -30515.367,E2 -30515.367} C_VEL
LIN {X 0,Y 22.835,Z 527.38,A -85,B 0,C 180,E1 -30529.942,E2 -30529.942} C_VEL
LIN {X 0,Y 23.648,Z 526.762,A -85,B 0,C 180,E1 -30534.175,E2 -30534.175} C_VEL
LIN {X 0,Y 30.712,Z 522.363,A -85,B 0,C 180,E1 -30553.366,E2 -30553.366} C_VEL
LIN {X 0,Y 40.568,Z 516.057,A -85,B 0,C 180,E1 -30565.387,E2 -30565.387} C_VEL
LIN {X 0,Y 49.788,Z 509.209,A -85,B 0,C 180,E1 -30571.925,E2 -30571.925} C_VEL
LIN {X 0,Y 59.379,Z 500.654,A -85,B 0,C 180,E1 -30576.541,E2 -30576.541} C_VEL
LIN {X 0,Y 67.624,Z 491.857,A -85,B 0,C 180,E1 -30579.295,E2 -30579.295} C_VEL
LIN {X 0,Y 75.978,Z 481.026,A -85,B 0,C 180,E1 -30581.476,E2 -30581.476} C_VEL
LIN {X 0,Y 82.689,Z 470.119,A -85,B 0,C 180,E1 -30582.986,E2 -30582.986} C_VEL
LIN {X 0,Y 88.781,Z 457.366,A -85,B 0,C 180,E1 -30584.335,E2 -30584.335} C_VEL
LIN {X 0,Y 92.971,Z 445.757,A -85,B 0,C 180,E1 -30585.107,E2 -30585.107} C_VEL
LIN {X 0,Y 96.164,Z 432.956,A -85,B 0,C 180,E1 -30585.72,E2 -30585.72} C_VEL
LIN {X 0,Y 97.887,Z 421.566,A -85,B 0,C 180,E1 -30586.161,E2 -30586.161} C_VEL
LIN {X 0,Y 97.422,Z 419.331,A -85,B 0,C 180,E1 -30589.609,E2 -30589.609} C_VEL
LIN {X 0,Y 97.246,Z 417.145,A -85,B 0,C 180,E1 -30595.855,E2 -30595.855} C_VEL
LIN {X 0,Y 97.483,Z 419.524,A -85,B 0,C 180,E1 -30601.265,E2 -30601.265} C_VEL
LIN {X 0,Y 97.911,Z 421.732,A -85,B 0,C 180,E1 -30604.372,E2 -30604.372} C_VEL
LIN {X 0,Y 95.795,Z 435.601,A -85,B 0,C 180,E1 -30604.818,E2 -30604.818} C_VEL
LIN {X 0,Y 92.566,Z 447.928,A -85,B 0,C 180,E1 -30605.312,E2 -30605.312} C_VEL
LIN {X 0,Y 88.33,Z 459.414,A -85,B 0,C 180,E1 -30605.948,E2 -30605.948} C_VEL
LIN {X 0,Y 82.287,Z 471.748,A -85,B 0,C 180,E1 -30606.819,E2 -30606.819} C_VEL
LIN {X 0,Y 76.273,Z 481.495,A -85,B 0,C 180,E1 -30607.865,E2 -30607.865} C_VEL
LIN {X 0,Y 68.618,Z 491.716,A -85,B 0,C 180,E1 -30609.641,E2 -30609.641} C_VEL
LIN {X 0,Y 59.377,Z 501.742,A -85,B 0,C 180,E1 -30612.431,E2 -30612.431} C_VEL
LIN {X 0,Y 50.297,Z 509.902,A -85,B 0,C 180,E1 -30616.226,E2 -30616.226} C_VEL
LIN {X 0,Y 40.126,Z 517.596,A -85,B 0,C 180,E1 -30623.127,E2 -30623.127} C_VEL
LIN {X 0,Y 32.852,Z 522.396,A -85,B 0,C 180,E1 -30631.146,E2 -30631.146} C_VEL
LIN {X 0,Y 25.43,Z 526.993,A -85,B 0,C 180,E1 -30646.283,E2 -30646.283} C_VEL
LIN {X 0,Y 20.894,Z 530.479,A -85,B 0,C 180,E1 -30670.332,E2 -30670.332} C_VEL
LIN {X 0,Y 20.339,Z 532.205,A -85,B 0,C 180,E1 -30689.987,E2 -30689.987} C_VEL
LIN {X 0,Y 20.929,Z 533.446,A -85,B 0,C 180,E1 -30709.609,E2 -30709.609} C_VEL
LIN {X 0,Y 23.595,Z 534.295,A -85,B 0,C 180,E1 -30726.55,E2 -30726.55} C_VEL
LIN {X 0,Y 27.789,Z 534.751,A -85,B 0,C 180,E1 -30739.337,E2 -30739.337} C_VEL
LIN {X 0,Y 38.811,Z 534.447,A -85,B 0,C 180,E1 -30754.862,E2 -30754.862} C_VEL
LIN {X 0,Y 51.431,Z 532.637,A -85,B 0,C 180,E1 -30763.031,E2 -30763.031} C_VEL
LIN {X 0,Y 59.062,Z 530.805,A -85,B 0,C 180,E1 -30766.234,E2 -30766.234} C_VEL
LIN {X 0,Y 71.421,Z 526.779,A -85,B 0,C 180,E1 -30769.726,E2 -30769.726} C_VEL
LIN {X 0,Y 81.661,Z 522.32,A -85,B 0,C 180,E1 -30771.756,E2 -30771.756} C_VEL
LIN {X 0,Y 93.733,Z 515.619,A -85,B 0,C 180,E1 -30773.424,E2 -30773.424} C_VEL
LIN {X 0,Y 104.128,Z 508.328,A -85,B 0,C 180,E1 -30774.554,E2 -30774.554} C_VEL
LIN {X 0,Y 114.577,Z 499.305,A -85,B 0,C 180,E1 -30775.355,E2 -30775.355} C_VEL
LIN {X 0,Y 122.167,Z 491.312,A -85,B 0,C 180,E1 -30775.838,E2 -30775.838} C_VEL
LIN {X 0,Y 126.791,Z 485.706,A -85,B 0,C 180,E1 -30776.113,E2 -30776.113} C_VEL
LIN {X 0,Y 126.774,Z 485.72,A -85,B 0,C 180,E1 -30776.227,E2 -30776.227} C_VEL
LIN {X 0,Y 117.862,Z 495.895,A -85,B 0,C 180,E1 -30777.135,E2 -30777.135} C_VEL
LIN {X 0,Y 108.99,Z 504.17,A -85,B 0,C 180,E1 -30778.087,E2 -30778.087} C_VEL
LIN {X 0,Y 98.393,Z 512.243,A -85,B 0,C 180,E1 -30779.382,E2 -30779.382} C_VEL
LIN {X 0,Y 87.86,Z 518.668,A -85,B 0,C 180,E1 -30781.029,E2 -30781.029} C_VEL
LIN {X 0,Y 77.412,Z 523.725,A -85,B 0,C 180,E1 -30783.037,E2 -30783.037} C_VEL
LIN {X 0,Y 65.133,Z 528.221,A -85,B 0,C 180,E1 -30786.196,E2 -30786.196} C_VEL
LIN {X 0,Y 56.933,Z 530.448,A -85,B 0,C 180,E1 -30789.081,E2 -30789.081} C_VEL
LIN {X 0,Y 50.315,Z 531.766,A -85,B 0,C 180,E1 -30792.131,E2 -30792.131} C_VEL
LIN {X 0,Y 37.725,Z 533.199,A -85,B 0,C 180,E1 -30801.353,E2 -30801.353} C_VEL
LIN {X 0,Y 31.967,Z 533.279,A -85,B 0,C 180,E1 -30808.447,E2 -30808.447} C_VEL
LIN {X 0,Y 22.817,Z 532.248,A -85,B 0,C 180,E1 -30831.987,E2 -30831.987} C_VEL
LIN {X 0,Y 20.452,Z 531.146,A -85,B 0,C 180,E1 -30849.915,E2 -30849.915} C_VEL
LIN {X 0,Y 21.582,Z 528.358,A -85,B 0,C 180,E1 -30882.31,E2 -30882.31} C_VEL
LIN {X 0,Y 23.648,Z 526.762,A -85,B 0,C 180,E1 -30894.175,E2 -30894.175} C_VEL
LIN {X 0,Y 26.277,Z 524.854,A -85,B 0,C 180,E1 -30905.524,E2 -30905.524} C_VEL
LIN {X 0,Y 30.849,Z 521.262,A -85,B 0,C 180,E1 -30921.75,E2 -30921.75} C_VEL
LIN {X 0,Y 36.825,Z 516.968,A -85,B 0,C 180,E1 -30933.181,E2 -30933.181} C_VEL
LIN {X 0,Y 41.236,Z 513.953,A -85,B 0,C 180,E1 -30936.979,E2 -30936.979} C_VEL
LIN {X 0,Y 51.888,Z 505.961,A -85,B 0,C 180,E1 -30941.477,E2 -30941.477} C_VEL
LIN {X 0,Y 60.331,Z 498.25,A -85,B 0,C 180,E1 -30943.969,E2 -30943.969} C_VEL
LIN {X 0,Y 69.757,Z 487.741,A -85,B 0,C 180,E1 -30945.878,E2 -30945.878} C_VEL
LIN {X 0,Y 77.48,Z 477.059,A -85,B 0,C 180,E1 -30947.202,E2 -30947.202} C_VEL
LIN {X 0,Y 83.475,Z 466.737,A -85,B 0,C 180,E1 -30948.179,E2 -30948.179} C_VEL
LIN {X 0,Y 88.821,Z 454.944,A -85,B 0,C 180,E1 -30949.031,E2 -30949.031} C_VEL
LIN {X 0,Y 93.13,Z 442.053,A -85,B 0,C 180,E1 -30949.63,E2 -30949.63} C_VEL
LIN {X 0,Y 95.985,Z 429.267,A -85,B 0,C 180,E1 -30950.037,E2 -30950.037} C_VEL
LIN {X 0,Y 96.396,Z 426.374,A -85,B 0,C 180,E1 -30950.207,E2 -30950.207} C_VEL
LIN {X 0,Y 96.348,Z 424.38,A -85,B 0,C 180,E1 -30955.816,E2 -30955.816} C_VEL
LIN {X 0,Y 96.409,Z 426.235,A -85,B 0,C 180,E1 -30959.999,E2 -30959.999} C_VEL
LIN {X 0,Y 96.429,Z 426.499,A -85,B 0,C 180,E1 -30960.393,E2 -30960.393} C_VEL
LIN {X 0,Y 93.809,Z 440.011,A -85,B 0,C 180,E1 -30960.736,E2 -30960.736} C_VEL
LIN {X 0,Y 90.049,Z 452.301,A -85,B 0,C 180,E1 -30961.127,E2 -30961.127} C_VEL
LIN {X 0,Y 85.232,Z 463.707,A -85,B 0,C 180,E1 -30961.532,E2 -30961.532} C_VEL
LIN {X 0,Y 79.122,Z 474.926,A -85,B 0,C 180,E1 -30962.084,E2 -30962.084} C_VEL
LIN {X 0,Y 72.143,Z 485.256,A -85,B 0,C 180,E1 -30963.041,E2 -30963.041} C_VEL
LIN {X 0,Y 65.182,Z 493.732,A -85,B 0,C 180,E1 -30964.122,E2 -30964.122} C_VEL
